// TwinCAT 3 PLC project HeatAndSteam
// ProgramVersion: 3.1.4023.0
// libraries:
//   Tc2_DataExchange, * (Beckhoff Automation GmbH)
//   Tc2_EtherCAT, * (Beckhoff Automation GmbH)
//   Tc2_MDP, * (Beckhoff Automation GmbH)
//   Tc2_ModbusSrv, * (Beckhoff Automation GmbH)
//   Tc2_Standard, * (Beckhoff Automation GmbH)
//   Tc2_SUPS, * (Beckhoff Automation GmbH)
//   Tc2_System, * (Beckhoff Automation GmbH)
//   Tc2_Utilities, * (Beckhoff Automation GmbH)
//   Tc3_DynamicMemory, * (Beckhoff Automation GmbH)
//   Tc3_EventLogger, * (Beckhoff Automation GmbH)
//   Tc3_Module, * (Beckhoff Automation GmbH)
//   Tc3_PackML_V2, * (Beckhoff Automation GmbH)
//   Tc3_PLCopen_OpcUa, * (Beckhoff Automation GmbH)
// project tree:
//   ECC/Basic/ADS Comm/ E_ADS_Comm_State.TcDUT, E_ADS_Comm_Type.TcDUT, FB_ADS_Comm.TcPOU
//   ECC/Basic/Cell/ FB_Cell_Basic.TcPOU, FB_PLC_Basic.TcPOU
//   ECC/Basic/Common Units/ E_Units.TcDUT, FB_Units.TcPOU
//   ECC/Basic/ GVL_BASIC.TcGVL
//   ECC/Basic/OPC Data/ E_StationJobData.TcDUT, F_NewDeviceDataX.TcPOU, ST_InputHeader.TcDUT, ST_OutputHeaderCellInformationX.TcDUT, ST_OutputHeaderMetaInformationX.TcDUT
//   ECC/Basic/OPC Data/Sub/ E_AlarmCategory.TcDUT, E_PML_Command.TcDUT, E_PML_Mode.TcDUT, E_PML_State.TcDUT, MaterialDataX.TcDUT, MaterialXMapping.TcDUT, ST_DataPointX.TcDUT, ST_DeviceDataX.TcDUT, ST_ErrorWarningDataX.TcDUT, ST_ManipulateMLX.TcDUT, ST_MaterialDataX.TcDUT, ST_OutputHeaderCellInformationStationInformationOperationInformationX.TcDUT, ST_OutputHeaderCellInformationStationX.TcDUT, ST_OutputHeaderTransportInformationX.TcDUT, ST_SKURestriction.TcDUT, ST_ToolDataX.TcDUT, ToolDataX.TcDUT, ToolX.TcDUT, ToolXMapping.TcDUT
//   ECC/Basic/OPC Data/Sub/Input/ ST_InputModeState.TcDUT
//   ECC/Basic/OPC Data/Sub/Output/ ST_Energy.TcDUT, ST_Exhaust.TcDUT, ST_Fluid.TcDUT, ST_JobDataOut.TcDUT, ST_OperationalDataOPxxxxx.TcDUT, ST_OutputErrorWarning.TcDUT, ST_OutputModeState.TcDUT, ST_OutputOEE.TcDUT
//   ECC/Basic/Station/ FB_Station_Basic.TcPOU
//   ECC/Basic/TrackClient/DUT/ E_CellType.TcDUT, E_MMDirection.TcTLEO, E_MMStationBuffer.TcTLEO, E_MMTrafficLightColor.TcTLEO, E_MMVehicleCommand.TcTLEO, E_MMVehicleInputType.TcTLEO, ST_MethodArgumentData.TcDUT, ST_MMBuffer.TcDUT, ST_MMLocation.TcDUT, ST_MMStation.TcDUT, ST_MMVehicleFlagData.TcDUT, ST_MMVehicleStatusData.TcDUT, ST_OPCUA_MethodData.TcDUT
//   ECC/Basic/TrackClient/Enums/ E_CarrierStatus.TcDUT, E_MMPathMotionStatus.TcTLEO, E_MMPathState.TcTLEO, E_MMServerStatus.TcTLEO, E_OPC_UA_Errors.TcDUT, E_TrackClientState.TcDUT, E_TrackState.TcDUT, E_VehicleMoveState.TcDUT
//   ECC/Basic/TrackClient/ E_CommandDataState.TcDUT, E_MappingDataState.TcDUT, E_ReworkDataState.TcDUT, FB_TrackClient_Basic.TcPOU
//   ECC/Basic/TrackClient/GVLs/ GlobalConstants.TcGVL
//   ECC/Basic/TrackClient/Method Data/Cell/ ST_GetCellIndexData.TcDUT, ST_GetCellIndexDataIn.TcDUT, ST_GetCellIndexDataOut.TcDUT
//   ECC/Basic/TrackClient/Method Data/Data/ E_MaterialType.TcDUT, E_ToolType.TcDUT, ST_AddReservationData.TcDUT, ST_AddReservationDataIn.TcDUT, ST_AddReservationDataOut.TcDUT, ST_RemoveReservationData.TcDUT, ST_RemoveReservationDataIn.TcDUT, ST_RemoveReservationDataOut.TcDUT, ST_UpdateStationBufferData.TcDUT, ST_UpdateStationBufferDataIn.TcDUT, ST_UpdateStationBufferDataOut.TcDUT, ST_UpdateVehicleDataData.TcDUT (excluded from build), ST_UpdateVehicleDataDataIn.TcDUT (excluded from build), ST_UpdateVehicleDataDataOut.TcDUT (excluded from build), ST_UpdateVehicleMappingDataData.TcDUT, ST_UpdateVehicleMappingDataDataIn.TcDUT, ST_UpdateVehicleMappingDataDataOut.TcDUT, ST_UpdateVehicleMontageData.TcDUT, ST_UpdateVehicleMontageDataIn.TcDUT, ST_UpdateVehicleMontageDataOut.TcDUT, ST_UpdateVehicleOwnerData.TcDUT, ST_UpdateVehicleOwnerDataIn.TcDUT, ST_UpdateVehicleOwnerDataOut.TcDUT, ST_UpdateVehicleReservationDataData.TcDUT, ST_UpdateVehicleReservationDataDataIn.TcDUT, ST_UpdateVehicleReservationDataDataOut.TcDUT, ST_UpdateVehicleReworkDataData.TcDUT, ST_UpdateVehicleReworkDataDataIn.TcDUT, ST_UpdateVehicleReworkDataDataOut.TcDUT
//   ECC/Basic/TrackClient/Method Data/MoveVehicle/ ST_MoveToBufferData.TcDUT, ST_MoveToBufferDataIn.TcDUT, ST_MoveToBufferDataOut.TcDUT, ST_MoveToDecisionPointData.TcDUT, ST_MoveToDecisionPointDataIn.TcDUT, ST_MoveToDecisionPointDataOut.TcDUT, ST_MoveToPositionData.TcDUT, ST_MoveToPositionDataIn.TcDUT, ST_MoveToPositionDataOut.TcDUT, ST_MoveToScannerData.TcDUT, ST_MoveToScannerDataIn.TcDUT, ST_MoveToScannerDataOut.TcDUT, ST_MoveToStationDataIn.TcDUT, ST_MoveToStationDataOut.TcDUT, ST_MoveToStationInData.TcDUT, ST_MoveToStationOutData.TcDUT, ST_MoveVehicleStatusData.TcDUT, ST_MoveVehicleStatusDataIn.TcDUT, ST_MoveVehicleStatusDataOut.TcDUT
//   ECC/Basic/TrackClient/Method Data/Path/ ST_AddPathData.TcDUT, ST_AddPathDataIn.TcDUT, ST_AddPathDataOut.TcDUT, ST_RemovePathData.TcDUT, ST_RemovePathDataIn.TcDUT, ST_RemovePathDataOut.TcDUT, ST_ResetPathData.TcDUT, ST_ResetPathDataIn.TcDUT, ST_ResetPathDataOut.TcDUT, ST_ResumePathData.TcDUT, ST_ResumePathDataIn.TcDUT, ST_ResumePathDataOut.TcDUT, ST_StartPathData.TcDUT, ST_StartPathDataIn.TcDUT, ST_StartPathDataOut.TcDUT, ST_SuspendPathData.TcDUT, ST_SuspendPathDataIn.TcDUT, ST_SuspendPathDataOut.TcDUT
//   ECC/Basic/TrackClient/Method Data/Segment/ ST_AddPathSegmentData.TcDUT, ST_AddPathSegmentDataIn.TcDUT, ST_AddPathSegmentDataOut.TcDUT, ST_GetPathSegmentVehicleCountData.TcDUT, ST_GetPathSegmentVehicleCountDataIn.TcDUT, ST_GetPathSegmentVehicleCountDataOut.TcDUT, ST_RemovePathSegmentData.TcDUT, ST_RemovePathSegmentDataIn.TcDUT, ST_RemovePathSegmentDataOut.TcDUT
//   ECC/Basic/TrackClient/Method Data/Station/ ST_AddStationData.TcDUT, ST_AddStationDataIn.TcDUT, ST_AddStationDataOut.TcDUT, ST_AddStationDoubleData.TcDUT, ST_AddStationDoubleDataIn.TcDUT, ST_AddStationDoubleDataOut.TcDUT, ST_AddStationSingleData.TcDUT, ST_AddStationSingleDataIn.TcDUT, ST_AddStationSingleDataOut.TcDUT, ST_AdjustBufferPosData.TcDUT, ST_AdjustBufferPosDataIn.TcDUT, ST_AdjustBufferPosDataOut.TcDUT, ST_EnableStationData.TcDUT, ST_EnableStationDataIn.TcDUT, ST_EnableStationDataOut.TcDUT, ST_RemoveStationData.TcDUT, ST_RemoveStationDataIn.TcDUT, ST_RemoveStationDataOut.TcDUT
//   ECC/Basic/TrackClient/Method Data/TrafficLight/ ST_AddTrafficLightData.TcDUT, ST_AddTrafficLightDataIn.TcDUT, ST_AddTrafficLightDataOut.TcDUT, ST_RemoveTrafficLightData.TcDUT, ST_RemoveTrafficLightDataIn.TcDUT, ST_RemoveTrafficLightDataOut.TcDUT, ST_SetTrafficLightColorData.TcDUT, ST_SetTrafficLightColorDataIn.TcDUT, ST_SetTrafficLightColorDataOut.TcDUT, ST_TrafficLightColorData.TcDUT, ST_TrafficLightColorDataIn.TcDUT, ST_TrafficLightColorDataOut.TcDUT
//   ECC/Basic/TrackClient/Node Data/ E_OPC_NodeType.TcDUT, ST_ReadCellData.TcDUT, ST_ReadNodeData.TcDUT, ST_ReadPathData.TcDUT, ST_ReadPathData_OLD.TcDUT, ST_ReadStationData.TcDUT, ST_ReadVehicleData.TcDUT, ST_ReadVehicleData_OLD.TcDUT, ST_StatusCell.TcDUT, ST_StatusNode.TcDUT, ST_StatusPath.TcDUT, ST_StatusStation.TcDUT, ST_StatusVehicle.TcDUT
//   ECC/Basic/TrackClient/Node Data/SUB/ ST_ReservationData.TcDUT
//   ECC/Basic/TrackClient/OPC Data/ ST_InputTransport.TcDUT, ST_OutputTransport.TcDUT
//   ECC/Basic/TrackClient/OPC Data/Sub/ ST_BufferIndexX.TcDUT, ST_CarrierX.TcDUT, ST_InputTransportAdditionalData.TcDUT, ST_InputTransportAdditionalDataMESHandShake.TcDUT, ST_InputTransportAdditionalDataSettings.TcDUT, ST_InputTransportCommand.TcDUT, ST_InputTransportConfiguration.TcDUT, ST_InputTransportMapping.TcDUT, ST_OutputTransportAdditionalData.TcDUT, ST_OutputTransportConfiguration.TcDUT, ST_OutputTransportMapping.TcDUT, ST_OutputTransportStatus.TcDUT, ST_StationBufferStatus.TcDUT, ST_StationBufferX.TcDUT, ST_StationConfigX.TcDUT, ST_StatusBuffer.TcDUT, ST_TrackLocation.TcDUT, ST_TransportMappingCarrier.TcDUT, ST_TransportMappingStationBuffer.TcDUT
//   ECC/Cell_Unit_4/ E_VehicleOnStation.TcDUT, FB_Cell_Unit_4.TcPOU, FB_OPC_Cell_Unit_4.TcPOU, ST_VehicleInHS.TcDUT
//   ECC/Cell_Unit_4/HeatAndSteamDeviceDriver/ FB_EMS_HS.TcPOU, U_EMS_HS_Read.TcDUT, U_EMS_HS_Write.TcDUT
//   ECC/Cell_Unit_4/HeatAndSteamDeviceDriver/Sub/ E_EMS_HS_Status.TcDUT, ST_EMS_HS_Alarms.TcDUT, ST_EMS_HS_Command.TcDUT, ST_EMS_HS_Read.TcDUT, ST_EMS_HS_States.TcDUT, ST_EMS_HS_Write.TcDUT
//   ECC/Cell_Unit_4/HeatAndSteam/ FB_HeatAndSteamOUT.TcPOU, F_CalcValuesHeatSteam.TcPOU, stStationVehicleCmdOut.TcDUT, E_HSStationINSeq.TcDUT, FB_HeatAndSteamIN.TcPOU
//   ECC/Cell_Unit_4/HeatAndSteam/OPC Data/Sub/AdditionalData/ ST_InputStationHSAdditionalDataOP11600.TcDUT, ST_InputStationHSAdditionalDataOP11601.TcDUT, ST_InputStationHSAdditionalDataMESHandShake.TcDUT, ST_InputStationHSAdditionalDataSettings.TcDUT, ST_OuputStationHSAdditionalDataOP11600.TcDUT, ST_OuputStationHSAdditionalDataOP11601.TcDUT, ST_InputStationHSAdditionalData.TcDUT, ST_InputStationHSAdditionalDataGeneral.TcDUT, ST_OutputStationHSAdditionalData.TcDUT, ST_OutputStationHSAdditionalDataGeneral.TcDUT
//   ECC/Cell_Unit_4/HeatAndSteam/OPC Data/Sub/Configuration/ ST_InputStationHSConfigurationOP11600.TcDUT, ST_InputStationHSUpcomingConfigurationOP11601.TcDUT, ST_InputStationHSConfigurationOP11601.TcDUT, ST_OutputStationHSCurrentConfigurationOP11601.TcDUT, ST_OutputStationHSUpcomingConfigurationOP11601.TcDUT, ST_InputStationHSConfiguration.TcDUT, ST_InputStationHSConfigurationGeneral.TcDUT, ST_InputStationHSUpcomingConfiguration.TcDUT, ST_InputStationHSUpcomingConfigurationOP11600.TcDUT, ST_OutputStationHSConfigurationOP11600.TcDUT, ST_OutputStationHSCurrentConfiguration.TcDUT, ST_OutputStationHSCurrentConfigurationGeneral.TcDUT, ST_OutputStationHSCurrentConfigurationOP11600.TcDUT, ST_OutputStationHSUpcomingConfiguration.TcDUT, ST_OutputStationHSUpcomingConfigurationOP11600.TcDUT
//   ECC/Cell_Unit_4/HeatAndSteam/OPC Data/Sub/Control/ ST_InputStationHSControlOP11601.TcDUT, ST_InputStationHSControl.TcDUT, ST_InputStationHSControlGeneral.TcDUT, ST_InputStationHSControlOP11600.TcDUT
//   ECC/Cell_Unit_4/HeatAndSteam/OPC Data/Sub/JobData/ ST_OutputStationHSJobDataOP11600.TcDUT, ST_InputStationHSJobDataOP11601.TcDUT, ST_OutputStationHSJobDataOP11601.TcDUT, ST_InputStationHSJobData.TcDUT, ST_InputStationHSJobDataOP11600.TcDUT, ST_OutputStationHSJobData.TcDUT
//   ECC/Cell_Unit_4/HeatAndSteam/OPC Data/Sub/OperationalData/ ST_OutputStationHSOperationalDataOP11601.TcDUT, ST_OutputStationHSOperationalData.TcDUT, ST_OutputStationHSOperationalDataGeneral.TcDUT, ST_OutputStationHSOperationalDataOP11600.TcDUT
//   ECC/Cell_Unit_4/OPC Data/ ST_Input.TcDUT, ST_Output.TcDUT
//   ECC/Cell_Unit_4/OPC Data/Sub/ ST_InputCell.TcDUT, ST_InputCellAdditionalData.TcDUT, ST_InputCellAdditionalDataMESHandShake.TcDUT, ST_InputCellAdditionalDataSettings.TcDUT, ST_InputCellConfiguration.TcDUT, ST_InputCellConfigurationGeneral.TcDUT, ST_InputCellControl.TcDUT, ST_InputStation.TcDUT, ST_OutputCell.TcDUT, ST_OutputCellAdditionalData.TcDUT, ST_OutputCellConfiguration.TcDUT, ST_OutputCellConfigurationGeneral.TcDUT, ST_OutputCellOperationalData.TcDUT, ST_OutputCellSustainabilityData.TcDUT, ST_OutputHeader.TcDUT, ST_OutputHeaderCellInformation.TcDUT, ST_OutputHeaderCellInformationStation.TcDUT, ST_OutputHeaderCellInformationStationInformationOperationInformation.TcDUT, ST_OutputStation.TcDUT, ST_OutputCellOperationalDataGeneral.TcDUT
//   ECC/Cell_Unit_4/HeatAndSteam/OPC Data/ ST_InputStationStationHS.TcDUT, ST_OutputStationStationHS.TcDUT
//   ECC/Cell_Unit_4/HeatAndSteam/OPC Data/Sub/Information/ ST_OutputHeaderCellInformationStationHS.TcDUT
//   ECC/Cell_Unit_4/HeatAndSteam/OPC Data/Sub/Sustainability/ ST_OutputStationHSSustainabilityData.TcDUT
//   ECC/Components/ E_ComponentErrors.TcDUT, E_Cylinder_Cmd.TcDUT, E_Cylinder_Sta.TcDUT, FB_AI.TcPOU, FB_AO.TcPOU, FB_Basic.TcPOU, FB_Blink.TcPOU, FB_Cylinder.TcPOU, FB_DI.TcPOU, FB_DO.TcPOU, FB_LIN_TRAFO.TcPOU, F_ECat_OK.TcPOU, GVL_Components.TcGVL
//   ECC/Components/TwinSAFE/ E_TwinSAFE_Group_Diag.TcDUT, E_TwinSAFE_Group_State.TcDUT, E_TwinSAFE_Logic_State.TcDUT, FB_TwinSAFE_Group.TcPOU
//   ECC/Tools/ E_Method.TcDUT, E_OPCUA_Client_Seq.TcDUT, FB_CheckHeartBeat.TcPOU, FB_GenerateHeartBeat.TcPOU, FB_GetCPULoad.TcPOU, FB_GetCPULoadPLC.TcPOU, FB_GetCPUTemp.TcPOU, FB_GetIPCSerial.TcPOU, FB_GetSafetyTemp.TcPOU, FB_GetTimePML.TcPOU, FB_OPCUA_Client_Basic.TcPOU, FB_OPCUA_Client_CallMethod.TcPOU, FB_OPCUA_Client_ReadVar.TcPOU, FB_OPCUA_GetRecipe.TcPOU, FB_OPCUA_ReadVar_BAK.TcPOU, F_Array_Sort.TcPOU, F_LogLine.TcPOU, F_StringCompNoCase.TcPOU, ST_OPC_Client_Data.TcDUT, ST_OutputArgInfoAndData_Basis.TcDUT, ST_Test.TcDUT
//   ECC/Tools/LogToFile/ FB_GetFifo.TcPOU, FB_LogToFile.TcPOU, FB_SetFifo.TcPOU, F_LogFile.TcPOU, F_PadWith.TcPOU, GVL_Log.TcGVL, ST_String_FIFO.TcDUT
//   ECC/TrackClient/Buffer Control/ FB_BufferControl.TcPOU, ST_BufferControl.TcDUT
//   ECC/TrackClient/Enums/ E_BufferState.TcDUT, E_BufferStates.TcDUT, E_PostBufferInState.TcDUT, E_DecisionPointState.TcDUT, E_ExitPointState.TcDUT, E_StationState.TcDUT, E_PostBufferOutState.TcDUT
//   ECC/TrackClient/ FB_TrackClient.TcPOU
//   ECC/TrackClient/Station Control/ E_StationBufferState.TcDUT, E_StationInOutState.TcDUT, FB_StationControl.TcPOU, ST_StationControlData.TcDUT
//   GVLs/ GVL.TcGVL
//   / PlcTask.TcTTO
//   POUs/ MAIN.TcPOU
//   ReadConfigFile/ DUT_STRUCT_VARIABLES.TcDUT, FB_ReadFile.TcPOU
// real-time tasks:
//   TASK PlcTask: cycle T#10ms, priority 20, ADS port 350
// I/O:
//   DEVICE PCI (EtherCAT) (disabled), AmsNetId 10.128.16.81.2.1
//     BusCoupler (EK1200) [EK1200-5000 EtherCAT Power supply (2A E-Bus)]
//       License (EL6070-0033) [EL6070-0033 1Ch. Licence key terminal, individual licences]
//       End (EL9011) [EL9011 End Terminal]
// variable links:
//   HeatAndSteam/HeatAndSteam Instance <-> PCI (EtherCAT)/BusCoupler (EK1200)/License (EL6070-0033)
//     PlcTask Inputs/MAIN.fbUnit4.License_AdsAdrr <-> InfoData/AdsAddr
//     PlcTask Inputs/MAIN.fbUnit4.License_State <-> InfoData/State
//     PlcTask Inputs/MAIN.fbUnit4.fbSafetyTemp.sSafetyNetID/port <-> InfoData/AdsAddr/port

CONFIGURATION HeatAndSteam
    RESOURCE PLC ON TwinCAT3
        TASK PlcTask(INTERVAL := T#10ms, PRIORITY := 20);
        PROGRAM MAIN WITH PlcTask : MAIN;
    END_RESOURCE
END_CONFIGURATION

// ---- ECC/Basic/ADS Comm/E_ADS_Comm_State.TcDUT
{attribute 'qualified_only'}
{attribute 'strict'}
TYPE E_ADS_Comm_State :
(
	Disabled := 0,
	Idle,
	Wait_Write,
	Writing,
	Write_Error,
	Wait_Read,
	Reading,
	Read_Error
);
END_TYPE

// ---- ECC/Basic/ADS Comm/E_ADS_Comm_Type.TcDUT
{attribute 'strict'}
TYPE E_ADS_Comm_Type :
(
	ADS_RD_FAST := 0,
	ADS_RD_SLOW,
	ADS_WR_FAST,
	ADS_WR_SLOW,
	ADS_RD_TRIG1,
	ADS_RD_TRIG2,
	ADS_RD_TRIG3,
	ADS_WR_TRIG1,
	ADS_WR_TRIG2,
	ADS_WR_TRIG3
);
END_TYPE

// ---- ECC/Basic/Common Units/E_Units.TcDUT
{attribute 'qualified_only'}
{attribute 'strict'}
// NOTE: Must match the array in FB_CommonUnits
TYPE E_Units :
(
	None := 0,	// 

	_m,			// Meter
	_cm,		// Centimeter
	_mm,		// Millimeter
	_um,		// Micrometer
	_nm,		// Nanometer
	
	_kg,		// Kilogram
	_g,			// Gram
	
	_RPM,		// RPM
	_mm_s,		// Millimeter pr. second
	_mm_min,	// Millimeter pr. minute
	_m_s,		// Meter pr. second
	_m_min,		// Meter pr. minute
	
	_mm_s_s,	// Millimeter pr second squared
	
	_pct,		// percent
	
	_deg,		// Degrees (angle)
	_degC,		// Degrees celcius
	_degF,		// Degrees fahrenheit
	
	_bar,		// Bar
	
	_day,		// day
	_hour,		// Hour
	_min,		// minute
	_s,			// Second
	_ms,		// Millisecond
	_us,		// Microsecond
	_ns,		// Nanosecond

	_Vac,		// Volt AC
	_Vdc,		// Volt DC
	_mV,		// Millivolt
	_a,			// Ampere
	_mA,		// Milliampere
	_uA,		// Microampere
	_KWh,		// Kilowatt hour
	_KW,		// Kilowatt
	_W,			// Watt
	_mW,		// Milliwatt
	_uW,		// Microwatt
	
	_MHz,		// Megahertz
	_kHz,		// Kilehertz
	_Hz,		// Hertz
	
	last
);
END_TYPE

// ---- ECC/Basic/OPC Data/E_StationJobData.TcDUT
{attribute 'strict'}
//
//	MAX number is 9!!
//
TYPE E_StationJobData :
(
	// Back Moulding
//	OP00100_			:= 0,

	// Brazilian Blocking
//	OP00200_			:= 0,

	// Strobeling
//	OP00300_			:= 0,

	// Manual Lasting
//	OP11400_			:= 0,

	// Automatic Lasting
//	OP11500_			:= 0,

	// Upper heat setting
//	OP11600_			:= 0,

	// Shank Placement
//	OP11700_			:= 0,

	// Ironing
//	OP11800_			:= 0,

	// Strobel Pressing
//	OP11900_			:= 0,

	// Blow Drying
//	OP12000_			:= 0,

	// Hammering
//	OP12100_			:= 0,

	// Filler Foam Placement
//	OP12200_			:= 0,

	// Manual Roughing
//	OP12300_			:= 0,

	// Robot Laser Roughing
//	OP12400_			:= 0,

	// Robot Mechanical Roughing
	OP12500_Motor 		:= 0,
	OP12500_Speed 		:= 1,
	OP12500_Pressure	:= 2,
	
	// Thread Burning
	OP12600_Heat		:= 0,
	OP12600_Air			:= 1,
	
	// Last Sorting
//	OP12700_			:= 0,

	// Last Handling
//	OP12800_			:= 0,

	// Sole Cooling
//	OP12900_			:= 0,

	// Sole Heating
//	OP13000_			:= 0,

	// Continouos Spraying
	OP13100_Color		:= 0,
	OP13100_SprayWidth	:= 1,
	OP13100_SprayPress	:= 2,
	OP13100_Tank1Press	:= 3,
	OP13100_Tank2Press	:= 4,
	
	// Burst Spraying
	OP13200_Color		:= 0,
	OP13200_SprayWidth	:= 1,
	OP13200_SprayPress	:= 2,
	OP13200_Tank1Press	:= 3,
	OP13200_Tank2Press	:= 4,
	OP13200_SprayTime	:= 5,
	OP13200_PauseTime	:= 6,

	// Sole Trimming
	OP13300_Speed		:= 0,
	OP13300_Amplitude	:= 1
	
	// Sole Buffing
//	OP13400_			:= 0,

	// Manual Delasting
//	OP13500_			:= 0,

	// Robot Delasting
//	OP13600_			:= 0,

	// Delacing
//	OP21900_			:= 0,

	// Injection
//	OP32800_			:= 0,

);
END_TYPE

// ---- ECC/Basic/OPC Data/ST_InputHeader.TcDUT
/// Standard Header for cells
TYPE ST_InputHeader :
STRUCT
	{attribute 'OPC.UA.DA.Description' := 'Header (0-100, 2 Hz)'}
	HeartBeat				: UINT;
END_STRUCT
END_TYPE

// ---- ECC/Basic/OPC Data/ST_OutputHeaderCellInformationX.TcDUT
TYPE ST_OutputHeaderCellInformationX :
STRUCT
	{attribute 'OPC.UA.DA.Description' := 'Cell name'}
	CellName				: STRING;

	{attribute 'OPC.UA.DA.Description' := 'CellID'}
	CellID					: STRING;

	{attribute 'OPC.UA.DA.Description' := 'Number of stations'}
	NumberOfStations		: UINT;

	{attribute 'OPC.UA.DA.Description' := 'Station information'}
	{attribute 'OPC.UA.DA.StructuredType' := '1'}
	TransportInformation	: ST_OutputHeaderTransportInformationX;

END_STRUCT
END_TYPE

// ---- ECC/Basic/OPC Data/ST_OutputHeaderMetaInformationX.TcDUT
TYPE ST_OutputHeaderMetaInformationX :
STRUCT
	{attribute 'OPC.UA.DA.Description' := 'Interface version'}
	InterfaceVersion		: UINT;

	{attribute 'OPC.UA.DA.Description' := 'PLC version'}
	PLCVersion				: UINT;

	{attribute 'OPC.UA.DA.Description' := 'Serial Number'}
	SerialNumber			: STRING;

	{attribute 'OPC.UA.DA.Description' := 'Cell type'}
	CellType				: STRING;

END_STRUCT
END_TYPE

// ---- ECC/Basic/OPC Data/Sub/E_AlarmCategory.TcDUT
{attribute 'qualified_only'}
TYPE E_AlarmCategory :
(
Configuration:= 1, 
Safety := 65536000,
TrackClient := 131072000,
OPCcomm := 196608000,
JobData := 262144000,
ConfigurationData := 327680000,
//GeneralSpare := 393216000,
//GeneralSpare := 458752000,
//GeneralSpare := 524288000,
//GeneralSpare := 589824000,
//GeneralSpare := 655360000,
OP11200 := 734003200,
OP11210 := 734658560,
OP11400 := 747110400,
OP11600 := 760217600,
OP11601 := 760283136,
OP11602 := 760348672,
OP11603 := 760414208,
OP11604 := 760479744,
OP11700 := 766771200,
OP12000 := 786432000,
OP12001 := 786497536,
OP12002 := 786563072,
OP12003 := 786628608,
OP12004 := 786694144,
OP12010 := 787087360,
OP12011 := 787152896,
OP12200 := 799539200,
OP12500 := 819200000,
OP12600 := 825753600,
OP12900 := 845414400,
OP12901 := 845479936,
OP12902 := 845545472,
OP12903 := 845611008,
OP12904 := 845676544,
OP12910 := 846069760,
OP12911 := 846135296,
OP12912 := 846200832,
OP12913 := 846266368,
OP12914 := 846331904,
OP13100 := 858521600,
OP13200 := 865075200,
OP13300 := 871628800,
OP13500 := 884736000,
OP13800 := 904396800,
OP16000 := 1048576000,
OP16100 := 1055129600,
OP16200 := 1061683200,
OP16300 := 1068236800,
OP16400 := 1074790400,
OP21900 := 1435238400,
OPSpare := 3276800000,
Robot := 3342336000,
LifterStation1Device := 3407872000,
LifterStation2Device := 3473408000,
LastingDevice := 3538944000
)UDINT;
END_TYPE

// ---- ECC/Basic/OPC Data/Sub/E_PML_Command.TcDUT
{attribute 'qualified_only'}
TYPE E_PML_Command :
(
	Undefined := 0,	// 0
	Reset,			// 1
	Start,			// 2
	Stop,			// 3
	Hold,			// 4
	Unhold,			// 5
	Suspend,		// 6
	Unsuspend,		// 7
	Abort,			// 8
	Clear,			// 9
	Complete		// 10
) UINT;
END_TYPE

// ---- ECC/Basic/OPC Data/Sub/E_PML_Mode.TcDUT
{attribute 'qualified_only'}
TYPE E_PML_Mode :
(
	Undefined := 0,		// Same as in E_PMLProtectedUnitMode in TC3_PackML_V2 library
	Production,			// Same as in E_PMLProtectedUnitMode in TC3_PackML_V2 library
	Maintenance,		// Same as in E_PMLProtectedUnitMode in TC3_PackML_V2 library
	Manual,				// Same as in E_PMLProtectedUnitMode in TC3_PackML_V2 library
	Calibration,		// ??
	Cleaning,			// ??
	Simulation			// Same as E_PMLProtectedUnitMode.Production, but with GVL_Components.bSIMUMode = TRUE
) UINT;
END_TYPE

// ---- ECC/Basic/OPC Data/Sub/E_PML_State.TcDUT
{attribute 'qualified_only'}
TYPE E_PML_State :
(
	Undefined := 0,	// 0
	Clearing,		// 1
	Stopped,		// 2
	Starting,		// 3
	Idle,			// 4
	Suspended,		// 5
	Execute,		// 6
	Stopping,		// 7
	Aborting,		// 8
	Aborted,		// 9
	Holding,		// 10
	Held,			// 11
	Unholding,		// 12
	Suspending,		// 13
	Unsuspending,	// 14
	Resetting,		// 15
	Completing,		// 16
	Complete		// 17
) UINT;
END_TYPE

// ---- ECC/Basic/OPC Data/Sub/Input/ST_InputModeState.TcDUT
TYPE ST_InputModeState :
STRUCT
	{attribute 'OPC.UA.DA.Description' := 'Change Request (0-255)'}
	ChangeRequest				: UINT;

	{attribute 'OPC.UA.DA.Description' := 'Requested mode (0-6)'}
	Mode						: UINT := E_PML_Mode.Production;

	{attribute 'OPC.UA.DA.Description' := 'Requested state (0-3,6,7,9'}
	State						: UINT;

END_STRUCT
END_TYPE

// ---- ECC/Basic/OPC Data/Sub/MaterialDataX.TcDUT
TYPE MaterialDataX :
STRUCT
	{attribute 'OPC.UA.DA.Description' := 'Type ID of material'}
	MaterialTypeID				: STRING(30);

	{attribute 'OPC.UA.DA.Description' := 'ID of location for material'}
	Location					: UINT;

	{attribute 'OPC.UA.DA.Description' := 'Indicator for material empty'}
	MaterialEmpty				: BOOL;

	{attribute 'OPC.UA.DA.Description' := 'Indicator for remaining material (%)'}
	MaterialRemaining			: BOOL;

END_STRUCT
END_TYPE

// ---- ECC/Basic/OPC Data/Sub/MaterialXMapping.TcDUT
TYPE MaterialXMapping :
STRUCT
	{attribute 'OPC.UA.DA.Description' := 'Type ID of material'}
	MaterialTypeID				: STRING(30);

	{attribute 'OPC.UA.DA.Description' := 'Location material is configured on'}
	Location					: UINT;

END_STRUCT
END_TYPE

// ---- ECC/Basic/OPC Data/Sub/Output/ST_Energy.TcDUT
TYPE ST_Energy :
STRUCT
END_STRUCT
END_TYPE

// ---- ECC/Basic/OPC Data/Sub/Output/ST_Exhaust.TcDUT
TYPE ST_Exhaust :
STRUCT
END_STRUCT
END_TYPE

// ---- ECC/Basic/OPC Data/Sub/Output/ST_Fluid.TcDUT
TYPE ST_Fluid :
STRUCT
END_STRUCT
END_TYPE

// ---- ECC/Basic/OPC Data/Sub/Output/ST_JobDataOut.TcDUT
TYPE ST_JobDataOut :
STRUCT
	{attribute 'OPC.UA.DA.Description' := 'Change Request (0-255)'}
	ChangeStatus				: UINT;
	
	{attribute 'OPC.UA.DA.Description' := 'Job data type'}
	JobDataType					: STRING(7);

	{attribute 'OPC.UA.DA.Description' := 'Job state (0: Undefined, 1: Idle, 2: Executing, 3: Completed'}
	JobState					: UINT;

END_STRUCT
END_TYPE

// ---- ECC/Basic/OPC Data/Sub/Output/ST_OperationalDataOPxxxxx.TcDUT
TYPE ST_OperationalDataOPxxxxx :
STRUCT
	{attribute 'OPC.UA.DA.Description' := 'Current number of tools where data is available'}
	NumberOfToolData			: UINT;

	{attribute 'OPC.UA.DA.Description' := 'Status variables for current operational data of tools'}
	{attribute 'OPC.UA.DA.StructuredType' := '1'}
	ToolData					: ARRAY [1..200] OF ToolDataX;

	{attribute 'OPC.UA.DA.Description' := 'Current number OF feeding material where data is available'}
	NumberOfMaterialData		: UINT;

	{attribute 'OPC.UA.DA.Description' := 'Status variables for current operational data of material'}
	{attribute 'OPC.UA.DA.StructuredType' := '1'}
	MaterialData				: ARRAY [1..200] OF MaterialDataX;

	{attribute 'OPC.UA.DA.Description' := 'Status variables for current operational data of devices'}
	{attribute 'OPC.UA.DA.StructuredType' := '1'}
	DeviceData					: ARRAY [1..200] OF ST_DeviceDataX;
	
END_STRUCT
END_TYPE

// ---- ECC/Basic/OPC Data/Sub/Output/ST_OutputErrorWarning.TcDUT
TYPE ST_OutputErrorWarning :
STRUCT
// Handshake part
	{attribute 'OPC.UA.DA.Description' := 'Change acknowledged (0-255)'}
	ChangeAcknowledge		: UINT;

	{attribute 'OPC.UA.DA.Description' := 'Change status (0-255)'}
	ChangeStatus			: UINT;

// Data part	
	{attribute 'OPC.UA.DA.Description' := 'Data has changed (0-65536)'}
	DataChange				: UINT;
	
	{attribute 'OPC.UA.DA.Description' := 'Current number of warnings'}
	NumberOfWarnings		: UINT;
		
	{attribute 'OPC.UA.DA.Description' := 'Current number of errors'}
	NumberOfErrors			: UINT;
	
	{attribute 'OPC.UA.DA.Description' := 'Current types of error/warnings'}
	{attribute 'OPC.UA.DA.StructuredType' := '1'}
	ErrorWarningData		: ARRAY [1..255] OF ST_ErrorWarningDataX;
	
END_STRUCT
END_TYPE

// ---- ECC/Basic/OPC Data/Sub/Output/ST_OutputModeState.TcDUT
TYPE ST_OutputModeState :
STRUCT
// Handshake part
	{attribute 'OPC.UA.DA.Description' := 'Change acknowledged (0-255)'}
	ChangeAcknowledge		: UINT;

	{attribute 'OPC.UA.DA.Description' := 'Change status (0-255)'}
	ChangeStatus			: UINT;

// Data part	
	{attribute 'OPC.UA.DA.Description' := 'Mode State data changed'}
	DataChange				: UINT;

	{attribute 'OPC.UA.DA.Description' := 'Mode State response (0-3)'}
	ModeStateResponse		: UINT;		// 0: Undefined, 1: Could not handle, 2: Request declined, 3: OK

	{attribute 'OPC.UA.DA.Description' := 'Current mode (0-6)'}
	CurrentMode				: UINT;

	{attribute 'OPC.UA.DA.Description' := 'Requested mode (0-6)'}
	RequestedMode			: UINT;

	{attribute 'OPC.UA.DA.Description' := 'Current state (0-17)'}
	CurrentState			: UINT;

	{attribute 'OPC.UA.DA.Description' := 'Requested state (0-17)'}
	RequestedState			: UINT;

END_STRUCT
END_TYPE

// ---- ECC/Basic/OPC Data/Sub/Output/ST_OutputOEE.TcDUT
TYPE ST_OutputOEE :
STRUCT
// Handshake part
	{attribute 'OPC.UA.DA.Description' := 'Change acknowledged (0-255)'}
	ChangeAcknowledge	: UINT;

	{attribute 'OPC.UA.DA.Description' := 'Change status (0-255)'}
	ChangeStatus		: UINT;

// Data part	
	{attribute 'OPC.UA.DA.Description' := 'Data has changed (0-65536)'}
	DataChange			: UINT;
	
	{attribute 'OPC.UA.DA.Description' := 'Date and time'}
	DateTime	 		: DT;
	
	{attribute 'OPC.UA.DA.Description' := ''}
	EventID		 		: UDINT;
	
	{attribute 'OPC.UA.DA.Description' := 'Counter for all processed products'}
	ProcessedProduct	: UDINT;

	{attribute 'OPC.UA.DA.Description' := 'Counter for all processed good products'}
	GoodProduct			: UDINT;

	{attribute 'OPC.UA.DA.Description' := 'Counter for all processed rejected products'}
	RejectedProduct		: UDINT;

END_STRUCT
END_TYPE

// ---- ECC/Basic/OPC Data/Sub/ST_DataPointX.TcDUT
TYPE ST_DataPointX :
STRUCT
	X					: REAL;	// Point on shoe. X value.
	Y					: REAL;	// Point on shoe. Y value.
	Z					: REAL;	// Point on shoe. Z value.
	Q1					: REAL;	// Point on shoe. Quaternion scalar part
	Q2					: REAL;	// Point on shoe. Quaternion x vector part
	Q3					: REAL;	// Point on shoe. Quaternion y vector part
	Q4					: REAL;	// Point on shoe. Quaternion z vector part
	Speed				: REAL;	// Speed setting.
	Acceleration		: REAL;	// Acceleration setting
	Zone				: REAL;	// Zone setting
//	ExternalTCP			: UINT;	// ID of external TCP. This can be referencepoints for tools or otherpoints of interests.
	ExternalTCPOffsetX	: REAL;	// External TCP offset. X value.
	ExternalTCPOffsetY	: REAL;	// External TCP offset. Y value.
	ExternalTCPOffsetZ	: REAL;	// External TCP offset. Z value.
	ExternalTCPOffsetQ1	: REAL;	// External TCP offset. Quaternion scalar part
	ExternalTCPOffsetQ2	: REAL;	// External TCP offset. Quaternion x vector part
	ExternalTCPOffsetQ3	: REAL;	// External TCP offset. Quaternion y vector part
	ExternalTCPOffsetQ4	: REAL;	// External TCP offset. Quaternion z vector part
	Validate			: BOOL;	// Indicator that a validation from the bridge is required before moving to a point. Robot will move to a safepos untill validation is recieved from the bridge
	arDeviceParameters	: ARRAY [0..9] OF REAL;	// See "E_StationJobData" for array specification

END_STRUCT
END_TYPE

// ---- ECC/Basic/OPC Data/Sub/ST_DeviceDataX.TcDUT
TYPE ST_DeviceDataX :
STRUCT
	{attribute 'OPC.UA.DA.Description' := 'The ID of the specific device'}
	DeviceID			: STRING(30);

	{attribute 'OPC.UA.DA.Description' := 'The descriptive name of the device'}
	DeviceName			: STRING(30);

	{attribute 'OPC.UA.DA.Description' := 'The ID of the operational data'}
	DataID				: UDINT;

	{attribute 'OPC.UA.DA.Description' := 'The descriptive name of the operational data'}
	DataName			: STRING(30);

	{attribute 'OPC.UA.DA.Description' := 'The value of the operational data'}
	Value				: REAL;

	{attribute 'OPC.UA.DA.Description' := 'The ID code for the measuring unit'}
	UnitID				: STRING(30);

	{attribute 'OPC.UA.DA.Description' := 'The symbolic description of the measuring unit'}
	Unit				: STRING(30);

END_STRUCT
END_TYPE

// ---- ECC/Basic/OPC Data/Sub/ST_ErrorWarningDataX.TcDUT
TYPE ST_ErrorWarningDataX :
STRUCT
	{attribute 'OPC.UA.DA.Description' := 'Error/Warning type. 0: Undefined, 1: Warning, 2: Error'}
	ErrorWarningType	: UINT;
	
	{attribute 'OPC.UA.DA.Description' := 'Cell ID or Station ID'}
	LocationID			: STRING(30);
	
	{attribute 'OPC.UA.DA.Description' := 'Trigger data and time'}
	DateTime			: STRING;	

	{attribute 'OPC.UA.DA.Description' := 'ID of the error/warning'}
	ErrorWarningID		: UDINT;	

	{attribute 'OPC.UA.DA.Description' := 'ID of the specific device/tool (optional)'}
	DeviceID			: STRING(30);	

	{attribute 'OPC.UA.DA.Description' := 'Severity of the event. 0: Undefined, 1: Low, 2: High'}
	Severity			: UINT;	

	{attribute 'OPC.UA.DA.Description' := 'ID from the native device'}
	NativeID			: UDINT;	

	{attribute 'OPC.UA.DA.Description' := 'Message from the native device'}
	NativeMessage		: STRING(80);	

END_STRUCT
END_TYPE

// ---- ECC/Basic/OPC Data/Sub/ST_ManipulateMLX.TcDUT
TYPE ST_ManipulateMLX :
STRUCT
	iNumberOfDataPoint		: USINT;			// Indicator for how many OF the data points that are filled out.
	ScaleOriginX 			: REAL;				// Origin of scale point. X value.
	ScaleOriginY			: REAL;				// Origin of scale point. Y value.
	ScaleOriginZ			: REAL;				// Origin of scale point. Z value.
	ScaleOriginQ1			: REAL;				// Origin of scale point. Quaternion scalar part
	ScaleOriginQ2			: REAL;				// Origin of scale point. Quaternion x vector part
	ScaleOriginQ3			: REAL;				// Origin of scale point. Quaternion y vector part
	ScaleOriginQ4			: REAL;				// Origin of scale point. Quaternion z vector part
	ScaleFactorX			: REAL;				// Scale factor in x direction.
	ScaleFactorYZ			: REAL;				// Scale factor in y and z direction.
	CalibrationOffsetX		: REAL;				// Offset from calibration of machine last. X value.
	CalibrationOffsetY		: REAL;				// Offset from calibration of machine last. Y value.
	CalibrationOffsetZ		: REAL;				// Offset from calibration of machine last. Z value.
	CalibrationOffsetQ1		: REAL;				// Offset from calibration of machine last. Quaternion scalar part
	CalibrationOffsetQ2		: REAL;				// Offset from calibration of machine last. Quaternion x vector part
	CalibrationOffsetQ3		: REAL;				// Offset from calibration of shoe last. Quaternion y vector part
	CalibrationOffsetQ4		: REAL;				// Offset FROM calibration OF shoe last. Quaternion z vector part	
	aDataPoints				: ARRAY [0..199] OF ST_DataPointX;// Parameters for first point on shoe/machine last.
END_STRUCT
END_TYPE

// ---- ECC/Basic/OPC Data/Sub/ST_MaterialDataX.TcDUT
TYPE ST_MaterialDataX :
STRUCT
	{attribute 'OPC.UA.DA.Description' := 'Job data type'}

END_STRUCT
END_TYPE

// ---- ECC/Basic/OPC Data/Sub/ST_OutputHeaderCellInformationStationInformationOperationInformationX.TcDUT
TYPE ST_OutputHeaderCellInformationStationInformationOperationInformationX :
STRUCT
	{attribute 'OPC.UA.DA.Description' := 'Operation name'}
	OperationName			: STRING;

	{attribute 'OPC.UA.DA.Description' := 'Operation ID'}
	OperationID				: STRING;

END_STRUCT
END_TYPE

// ---- ECC/Basic/OPC Data/Sub/ST_OutputHeaderCellInformationStationX.TcDUT
TYPE ST_OutputHeaderCellInformationStationX :
STRUCT
	{attribute 'OPC.UA.DA.Description' := 'Station name'}
	StationName				: STRING;

	{attribute 'OPC.UA.DA.Description' := 'Station ID'}
	StationID				: STRING;
	
	{attribute 'OPC.UA.DA.Description' := 'PLC version'}
	NumberOfOperations		: UINT;
	
	{attribute 'OPC.UA.DA.Description' := 'Rework possible on this station'}
	Rework					: BOOL;

END_STRUCT
END_TYPE

// ---- ECC/Basic/OPC Data/Sub/ST_OutputHeaderTransportInformationX.TcDUT
TYPE ST_OutputHeaderTransportInformationX :
STRUCT
	{attribute 'OPC.UA.DA.Description' := 'Transport name'}
	TransportName			: STRING;

	{attribute 'OPC.UA.DA.Description' := 'Transport type'}
	TransportType			: STRING;
	
END_STRUCT
END_TYPE

// ---- ECC/Basic/OPC Data/Sub/ST_SKURestriction.TcDUT
TYPE ST_SKURestriction :
STRUCT
	{attribute 'OPC.UA.DA.Description' := 'TRUE of restrictions are active'}
	Restricted				: BOOL;

	{attribute 'OPC.UA.DA.Description' := 'Number of defined SKU restrictions (0-200)'}
	NumberOfRestrictions	: UINT;
	
	{attribute 'OPC.UA.DA.Description' := 'ID of SKUs that the operation is restricted to handle'}
	SKUID					: ARRAY [1..200] OF STRING(30);
	
END_STRUCT
END_TYPE

// ---- ECC/Basic/OPC Data/Sub/ST_ToolDataX.TcDUT
TYPE ST_ToolDataX :
STRUCT
	{attribute 'OPC.UA.DA.Description' := 'Job data type'}

END_STRUCT
END_TYPE

// ---- ECC/Basic/OPC Data/Sub/ToolDataX.TcDUT
TYPE ToolDataX :
STRUCT
	{attribute 'OPC.UA.DA.Description' := 'Unique ID of Tool'}
	TooID					: UINT;

	{attribute 'OPC.UA.DA.Description' := 'ID of the location of Tool'}
	Location				: UINT;

	{attribute 'OPC.UA.DA.Description' := 'Usage cycles since tool configuration'}
	CurrentCycles			: UDINT;

	{attribute 'OPC.UA.DA.Description' := 'Max allowed cycles for tool'}
	MaxCycles				: UDINT;

END_STRUCT
END_TYPE

// ---- ECC/Basic/OPC Data/Sub/ToolX.TcDUT
TYPE ToolX :
STRUCT
	{attribute 'OPC.UA.DA.Description' := 'Unique ID of tool'}
	ToolID					: STRING(30);
	
	{attribute 'OPC.UA.DA.Description' := 'ID for type of tool'}
	ToolTypeID				: STRING(30);

END_STRUCT
END_TYPE

// ---- ECC/Basic/OPC Data/Sub/ToolXMapping.TcDUT
TYPE ToolXMapping :
STRUCT
	{attribute 'OPC.UA.DA.Description' := 'Unique ID of tool'}
	ToolID						: STRING(30);

	{attribute 'OPC.UA.DA.Description' := 'ID for the location tool is configured on'}
	Location					: UINT;

	{attribute 'OPC.UA.DA.Description' := 'Max allowed tool cycles'}
	MaxCycles					: UINT;

END_STRUCT
END_TYPE

// ---- ECC/Basic/TrackClient/DUT/E_CellType.TcDUT
{attribute 'qualified_only'}
{attribute 'strict'}
TYPE E_CellType :
(
	Type_Outline := 0,		// Cell has own track with inlet and outlet tracks
	Type_Inline := 1,		// Cell/station is placed on the main track
	Type_InOut := 2			// Cell has only one track for handling both inlet and outlet (no queue functionality)
	
	
);
END_TYPE

// ---- ECC/Basic/TrackClient/DUT/E_MMDirection.TcTLEO
{attribute 'qualified_only'}
TYPE E_MMDirection :
(
	eMMDirection_BiDirectional	:= 0,																				(**)
	eMMDirection_Forward		:= 1,																				(**)
	eMMDirection_Backward		:= 2																				(**)
) BYTE;
END_TYPE

// ---- ECC/Basic/TrackClient/DUT/E_MMStationBuffer.TcTLEO
{attribute 'qualified_only'}
{attribute 'strict'}
TYPE E_MMStationBuffer :
(
	eMMStationBuffer_PreProcess		:= 0,
	eMMStationBuffer_PostProcess	:= 1
);
END_TYPE

// ---- ECC/Basic/TrackClient/DUT/E_MMTrafficLightColor.TcTLEO
{attribute 'qualified_only'}
TYPE E_MMTrafficLightColor :
(
	eMMTrafficLightColor_NA		:= -1,
	eMMTrafficLightColor_Green	:= 0,
	eMMTrafficLightColor_Red	:= 1
);
END_TYPE
//  eMMTrafficLightColor_NA = '-1'

// ---- ECC/Basic/TrackClient/DUT/E_MMVehicleCommand.TcTLEO
{attribute 'qualified_only'}
TYPE E_MMVehicleCommand :
(
	eMMVehicleCommand_NoCommandInProgress 	:= 0,																	(**)
	eMMVehicleCommand_MoveVehicleToStation	:= 176,																	(**)
	eMMVehicleCommand_MoveVehicleToPosition	:= 177																	(**)
) BYTE;
END_TYPE

// ---- ECC/Basic/TrackClient/DUT/E_MMVehicleInputType.TcTLEO
{attribute 'qualified_only'}
{attribute 'strict'}
TYPE E_MMVehicleInputType :
(
	eMMVehicleInputType_VehicleID			:= 0,	// MagneMotion ID
	eMMVehicleInputType_CarrierID			:= 1,	// RFID scanned ID from Carrier
	eMMVehicleInputType_LastID 				:= 2,	// RFID scanned Id from Last
	eMMVehicleInputType_ArticleID 			:= 3,
	eMMVehicleInputType_LastTypeID			:= 4,
	eMMVehicleInputType_StationID			:= 5,
	eMMVehicleInputType_CellID				:= 6,
	eMMVehicleInputType_EmptyVehicles		:= 7,
	eMMVehicleInputType_ReleasedVehicles	:= 8,
	eMMVehicleInputType_AllVehicles			:= 9
);
END_TYPE

// ---- ECC/Basic/TrackClient/DUT/ST_MethodArgumentData.TcDUT
TYPE ST_MethodArgumentData :
STRUCT
	eDataType		: E_UADataType;
	pData			: PVOID;
	nDataSize		: UINT;
	
END_STRUCT
END_TYPE

// ---- ECC/Basic/TrackClient/DUT/ST_MMBuffer.TcDUT
{attribute 'OPC.UA.DA.StructuredType':='1'}
TYPE ST_MMBuffer :
STRUCT
	bPresent					: BOOL	:= FALSE;																	(* Flag for indicating if the buffer position is present/used*)
	stLocation					: ST_MMLocation;																	(* Location of the buffer on the track. *)
	nTicket						: UINT;
	nTicketSize					: UINT;
	nReservedVehicleID			: UINT;
	nCurrentVehicleID			: UINT;
	CurrentPriority				: UINT;
//	sReservedCarrierID			: STRING(30);
//	sCurrentCarrierID			: STRING(30);
END_STRUCT
END_TYPE

// ---- ECC/Basic/TrackClient/DUT/ST_MMLocation.TcDUT
{attribute 'OPC.UA.DA.StructuredType':='1'}
TYPE ST_MMLocation :
STRUCT
	nPathID						: UINT	:= 0;		(* The path the position is related to. *)
	fPosition					: REAL	:= 0;		(* [M] The position on the path. *)
END_STRUCT
END_TYPE

// ---- ECC/Basic/TrackClient/DUT/ST_MMStation.TcDUT
{attribute 'OPC.UA.DA.StructuredType':='1'}
TYPE ST_MMStation :
STRUCT
	sCellID						: STRING := '';												(* The cell that the station belongs to. *)
	sStationID					: STRING(30) := '';											(* The identifier for the station. *)
	bPresent					: BOOL := FALSE;											(* Flag for indicating if the station is present. *)
	stStationData1				: ST_MMBuffer;												(* The location of the station. *)
	stStationData2				: ST_MMBuffer;												(* The location of the station. *)
	stDecisionLocation			: ST_MMLocation;											(* The location of the decision point of the station. *)
	astPreBuffer				: ARRAY[1..MM_MAX_BUFFER_INDEX] OF ST_MMBuffer;				(* The stations prebuffer. *)
	astPostBuffer				: ARRAY[1..MM_MAX_BUFFER_INDEX] OF ST_MMBuffer;				(* The stations postbuffer. *)
END_STRUCT
END_TYPE

// ---- ECC/Basic/TrackClient/DUT/ST_MMVehicleFlagData.TcDUT
TYPE ST_MMVehicleFlagData :
STRUCT
	bVehicleSignal				: BOOL;
	bObstructedStatus			: BOOL;
	bHinderedStatus				: BOOL;
	nPIDLoopSetIndex			: USINT;
	bSuspectStatus				: BOOL;
END_STRUCT
END_TYPE

// ---- ECC/Basic/TrackClient/DUT/ST_MMVehicleStatusData.TcDUT
TYPE ST_MMVehicleStatusData :
STRUCT
	nVehicleID					: UINT;
	bVehiclePresent				: BOOL;
	nPathID						: UINT;
	nDestinationPathID			: UINT;
	fVehiclePosition			: REAL;
	fVelocity					: REAL;
	eVehicleCommandType			: E_MMVehicleCommand;
	stVehicleFlags				: ST_MMVehicleFlagData;
	fVehicleCommandedPosition	: REAL;
	nVehicleCommandedStation	: USINT;
END_STRUCT
END_TYPE

// ---- ECC/Basic/TrackClient/DUT/ST_OPCUA_MethodData.TcDUT
// Data needed for OPC UA method calling
TYPE ST_OPCUA_MethodData :
STRUCT
	bActivate						: BOOL;		// TRUE to use this method call

	// Method information:
	sRemoteObjectName				: STRING;	// Remote object. e.g. 'MAIN.fbMMServer'
	sRemoteMethodName				: STRING;	// Remote method. e.g. 'M_AddPath'

	// Input data:
	NoOfInputArgs					: BYTE;		// Number of input arguments for the remote method
	
	
	// Output data:
	NoOfOutputArgs					: BYTE;		// Number of output arguments for the remote method
	
	
END_STRUCT
END_TYPE

// ---- ECC/Basic/TrackClient/Enums/E_CarrierStatus.TcDUT
{attribute 'qualified_only'}
{attribute 'strict'}
TYPE E_CarrierStatus :
(
	Undefined := 0,			// Recently discovered, not scanned or assigned to anything
	Initiating,				// On the way to scanning
	NotBusy,				// Not assigned to a job
	Busy,					// Assigned to a job
	MontageReserved			// Reserved for a tool, but tool is removed temporarily (must be free to mount same tool again)

);
END_TYPE

// ---- ECC/Basic/TrackClient/Enums/E_MMPathMotionStatus.TcTLEO
{attribute 'qualified_only'}
TYPE E_MMPathMotionStatus :
(
	eMMPathMotionStatus_Enabled				:= 0,																	(**)
	eMMPathMotionStatus_SuspendedByCommand	:= 1,																	(**)
	eMMPathMotionStatus_EStopActive			:= 2,																	(**)
	eMMPathMotionStatus_InterlockActive		:= 3																	(**)
) BYTE;
END_TYPE

// ---- ECC/Basic/TrackClient/Enums/E_MMPathState.TcTLEO
{attribute 'qualified_only'}
TYPE E_MMPathState :
(
	eMMPathState_Initialization 		:= 0,																		(**)
	eMMPathState_Startup				:= 1,																		(**)
	eMMPathState_Operational			:= 2,																		(**)
	eMMPathState_ResetInProgress		:= 3,																		(**)
	eMMPathState_ProgrammingInProgress	:= 4																		(**)
) BYTE;
END_TYPE

// ---- ECC/Basic/TrackClient/Enums/E_MMServerStatus.TcTLEO
{attribute 'qualified_only'}
{attribute 'strict'}
TYPE E_MMServerStatus :
(
	eMMServerStatus_Default										:= 0,
	eMMServerStatus_Success										:= 1,
	eMMServerStatus_Rejected_UserInputError						:= 2,
	eMMServerStatus_Rejected_NotAllowed							:= 3,
	eMMServerStatus_Rejected_ConfigurationAlreadyDefined		:= 20,
	eMMServerStatus_Rejected_NotDefinedInConfiguration			:= 21,
	eMMServerStatus_Rejected_VehicleRelatedInfoNotFound			:= 40,
	eMMServerStatus_Failed_UnableToRemoveFromConfiguration		:= 100,
	eMMServerStatus_Failed_CouldNotHandleMoveVehicleRequest		:= 120
);
END_TYPE

// ---- ECC/Basic/TrackClient/Enums/E_OPC_UA_Errors.TcDUT
{attribute 'qualified_only'}
TYPE E_OPC_UA_Errors :
(
	NO_ERROR						:= 16#00000000, // No error
	DEVICE_INVALIDSIZE				:= 16#00000705, // Parameter size not correct
	DEVICE_INVALIDDATA				:= 16#00000706, // Invalid parameter values
	DEVICE_NOMEMORY					:= 16#0000070A, // Not enough memory

	UAC_E_FAIL						:= 16#E4DD0001, // UA service call failed
	UAC_E_CONNECTED					:= 16#E4DD0100, // Server already connected
	UAC_E_CONNECT					:= 16#E4DD0101, // General error when establishing a connection
	UAC_E_UASECURITY				:= 16#E4DD0102, // UA security could not be set up
	UAC_E_ITEMEXISTS				:= 16#E4DD0103, // Element ID already exists
	UAC_E_ITEMNOTFOUND				:= 16#E4DD0104, // Element does not exist
	UAC_E_ITEMTYPE					:= 16#E4DD0105, // Invalid or unsupported item type
	UAC_E_CONVERSION				:= 16#E4DD0106, // Variable types cannot be converted
	UAC_E_SUSPENDED					:= 16#E4DD0107, // Device hangs. Please try again later...
	UAC_E_TYPE_NOT_SUPPORTED		:= 16#E4DD0108, // Conversion variable type is not supported.
	UAC_E_NSNAME_NOTFOUND			:= 16#E4DD0109, // No namespace with the specified name found.
	UAC_E_CONNECT_NOTFOUND			:= 16#E4DD0110, // Connection failed: Target host could not be found.
	UAC_E_TIMEOUT					:= 16#E4DD0111, // Timeout: i.e. target host does not respond
	UAC_E_INVALIDHDL				:= 16#E4DD0112, // Session handle invalid
	UAC_E_INVALIDNODEID				:= 16#E4DD0113, // UA node ID unknown
	UAC_E_INVAL_IDENTIFIER_TYPE		:= 16#E4DD0114, // Identifier type of UaNodeId invalid
	UAC_E_IDENTIFIER_NOTSUPP		:= 16#E4DD0115, // Identifier type UaNodeId is not supported
	UAC_E_INVAL_NODE_HDL			:= 16#E4DD0116, // Invalid node handle
	UAC_E_UAREADFAILED				:= 16#E4DD0117, // UA read failed for unknown reasons
	UAC_E_UAWRITEFAILED				:= 16#E4DD0118, // UA write failed for unknown reasons
	UAC_E_INVAL_NODEMETHOD_HDL		:= 16#E4DD0119, // Invalid method handle
	UAC_E_CALL_FAILED				:= 16#E4DD011A, // Call failed, cause unknown
	UAC_E_CALLDECODE_FAILED			:= 16#E4DD011B, // Successful call, decoding return value failed
	UAC_E_NOTMAPPEDTYPE				:= 16#E4DD011C, // Unassigned data type in return value
	UAC_E_CALL_FAILED_BADINTERNAL	:= 16#E4DD011D, // Call failed with UA_BadInternal
	UAC_E_METHODIDINVALID			:= 16#E4DD011E, // Unknown MethodID (returned on call, even if provided by GetMethodHdl)
	UAC_E_TOOMUCHDIM				:= 16#E4DD011F, // Method call has returned parameters with more than 3 dimensions; not supported.
	UAC_E_CALL_FAILED_INVALIDARG	:= 16#E4DD0120, // Call failed with OpcUa_BadInvalidArgument
	UAC_E_CALL_FAILED_TYPEMISMATCH	:= 16#E4DD0121, // Call failed with UAC_E_CALL_FAILED_TYPEMISMATCH
	UAC_E_CALL_FAILED_OUTOFRANGE	:= 16#E4DD0122, // Call failed with UAC_E_CALL_FAILED_OUTOFRANGE
	UAC_E_CALL_FAILED_BADSTRUCTURE	:= 16#E4DD0123, // Call failed with OpcUa_BadStructureMissing
	UAC_E_CALL_TYPEMISMATCH_OUTPARAM:= 16#E4DD0124, // Call successful, but type of output information provided does not match
	UAC_E_NONVALIDTYPEINFO			:= 16#E4DD0125, // Node has insufficient type information
	UAC_E_INVALIDATTRIBID			:= 16#E4DD0126, // Access to invalid node attribute
	UAC_E_NOTSUPPORTED				:= 16#E4DD0128, // The command is not supported by the connected UaServer, e.g. when calling UA_HistoryUpdate.
	UAC_E_INVALID_ARRAY_LENGTH		:= 16#E4DE0100, // An invalid array length not matching DataValueCount was assigned to UA_HistoryUpdate.
	UAC_E_INVALID_DATASIZE			:= 16#E4DE0101, // A data value with an invalid data type size was assigned to UA_HistoryUpdate. All assigned DataValues must be of the same data type.
	UAC_E_SUBERROR					:= 16#E4DE0102 // A lower-level error was output for at least one of the transferred data values. See ValueErrorIDs at UA_HistoryUpdate.
		
) UDINT;
END_TYPE

// ---- ECC/Basic/TrackClient/Enums/E_TrackClientState.TcDUT
{attribute 'qualified_only'}
{attribute 'strict'}
TYPE E_TrackClientState :
(
	Disconnected := 0,
	(* Connect *)
	Connecting,
	GetNamespaceIndex,
	Connected,
	(* Execute function *)
	GetHandle,
	Execute,
	ReleaseHandle,
	(* Disconnect *)	
	Disconnecting,
	Error
);
END_TYPE

// ---- ECC/Basic/TrackClient/Enums/E_TrackState.TcDUT
{attribute 'qualified_only'}
{attribute 'strict'}
TYPE E_TrackState :
(
	Undefined := 0,
	CheckInitDone,
//	InitDecisionPoint,
	WaitAllowInit,
	InitStations,
	SetPreBufferAdjust,
	SetPostBufferAdjust,
	InitPaths,
//	InitPathsStations,
//	InitPathsDecisionPoint,
//	InitPathsTrafficLight,
	InitGetCellIndex,
	Idle,
	Resetting,
	ResetWait,
	ResetCheck,
	Starting,
	StartCheck,
	InitTrafficLight,
	InitTrafficLight2,
	InitPathSegment,
	InitPathSegment2,
	InitVehicles,
	Started,
	Suspend,
	Suspending,
	Suspended,
	Resume,
	Resuming,
	Error
);
END_TYPE

// ---- ECC/Basic/TrackClient/Enums/E_VehicleMoveState.TcDUT
{attribute 'qualified_only'}
{attribute 'strict'}
TYPE E_VehicleMoveState :
(
	Unknown := 0,
	Idle,
	Pending,
	Accepted,
	Moving,
	Complete,
	ErrorLocation
	
);
END_TYPE

// ---- ECC/Basic/TrackClient/E_CommandDataState.TcDUT
{attribute 'qualified_only'}
{attribute 'strict'}
TYPE E_CommandDataState :
(
	Undefined := 0,
	CheckRequest,
	AddReservation,
	UpdateJobData,
	Done,
	Error
);
END_TYPE

// ---- ECC/Basic/TrackClient/E_MappingDataState.TcDUT
{attribute 'qualified_only'}
{attribute 'strict'}
TYPE E_MappingDataState :
(
	Undefined := 0,
	CheckRequest,
	UpdateMappingData,
	UpdateReworkData,
	Done,
	Error
);
END_TYPE

// ---- ECC/Basic/TrackClient/E_ReworkDataState.TcDUT
{attribute 'qualified_only'}
{attribute 'strict'}
TYPE E_ReworkDataState :
(
	Undefined := 0,
	CheckRequest,
	UpdateReworkData,
	Done,
	Error
);
END_TYPE

// ---- ECC/Basic/TrackClient/Method Data/Cell/ST_GetCellIndexData.TcDUT
TYPE ST_GetCellIndexData :
STRUCT
	sObjectID					: STRING := 'MAIN.fbMMServer';
	sMethodID					: STRING := 'MAIN.fbMMServer#M_GetCellIndex';
	iStatus						: INT;
	iNoOfInputArgs				: BYTE := 1;
	iNoOfOutputArgs				: BYTE := 3;
	stInput						: ST_GetCellIndexDataIn;
	stOutput					: ST_GetCellIndexDataOut;	
END_STRUCT
END_TYPE

// ---- ECC/Basic/TrackClient/Method Data/Cell/ST_GetCellIndexDataIn.TcDUT
{attribute 'pack_mode' := '1'}
TYPE ST_GetCellIndexDataIn :
STRUCT
	sCellID						: STRING(30);
END_STRUCT
END_TYPE

// ---- ECC/Basic/TrackClient/Method Data/Cell/ST_GetCellIndexDataOut.TcDUT
{attribute 'pack_mode' := '1'}
TYPE ST_GetCellIndexDataOut :
STRUCT
	// Fixed data for all methods
	nNumberOfOutputArguments	: UDINT;								// determined amount of output parameters
	nReserved					: ARRAY[1..4] OF BYTE;					// Reserved padding
	
	// Method specific data
	stOutputArgInfo				: ARRAY[1..3] OF ST_UAMethodArgInfo; 	//
	nCellIndex					: UINT; 								// Cell index for status structures on Track Server
	eStatus						: E_MMServerStatus;						// Status from remote method (succes/fail)
	sMessage					: STRING;								// Debugging message

END_STRUCT
END_TYPE

// ---- ECC/Basic/TrackClient/Method Data/Data/E_MaterialType.TcDUT
{attribute 'qualified_only'}
{attribute 'strict'}
TYPE E_MaterialType :
(
	Undefined := 0,
	None,
	Upper
);
END_TYPE

// ---- ECC/Basic/TrackClient/Method Data/Data/E_ToolType.TcDUT
{attribute 'qualified_only'}
{attribute 'strict'}
TYPE E_ToolType :
(
	Undefined := 0,
	None,
	Last,
	Tray
);
END_TYPE

// ---- ECC/Basic/TrackClient/Method Data/Data/ST_AddReservationData.TcDUT
TYPE ST_AddReservationData :
STRUCT
	sObjectID					: STRING := 'MAIN.fbMMServer';
	sMethodID					: STRING := 'MAIN.fbMMServer#M_AddReservationList';
	iStatus						: INT;
	iNoOfInputArgs				: BYTE := 5;
	iNoOfOutputArgs				: BYTE := 2;
	stInput						: ST_AddReservationDataIn;
	stOutput					: ST_AddReservationDataOut;	
END_STRUCT
END_TYPE

// ---- ECC/Basic/TrackClient/Method Data/Data/ST_AddReservationDataIn.TcDUT
{attribute 'pack_mode' := '1'}
TYPE ST_AddReservationDataIn :
STRUCT
	sStationID					: STRING(30);								(* The ID of the station that will be moved to. *)
	sCarrierID					: STRING(30);								(* Carrier ID of vehicle at buffer position *)
	nTicket						: UINT;										(* Ticket number *)
	nTicketSize					: UINT;										(* Ticket size (number of vehicles with same ticket) *)
	nPriority					: UINT;										(* Ticket priority *)
END_STRUCT
END_TYPE

// ---- ECC/Basic/TrackClient/Method Data/Data/ST_AddReservationDataOut.TcDUT
{attribute 'pack_mode' := '1'}
TYPE ST_AddReservationDataOut :
STRUCT
	// Fixed data for all methods
	nNumberOfOutputArguments	: UDINT;								// determined amount of output parameters
	nReserved					: ARRAY[1..4] OF BYTE;					// Reserved padding
	
	// Method specific data
	stOutputArgInfo				: ARRAY[1..2] OF ST_UAMethodArgInfo; 	// 
	eStatus						: E_MMServerStatus;						// Status from remote method (succes/fail)
	sMessage					: STRING;								// Debugging message

END_STRUCT
END_TYPE

// ---- ECC/Basic/TrackClient/Method Data/Data/ST_RemoveReservationData.TcDUT
TYPE ST_RemoveReservationData :
STRUCT
	sObjectID					: STRING := 'MAIN.fbMMServer';
	sMethodID					: STRING := 'MAIN.fbMMServer#M_RemoveReservationList';
	iStatus						: INT;
	iNoOfInputArgs				: BYTE := 2;
	iNoOfOutputArgs				: BYTE := 2;
	stInput						: ST_RemoveReservationDataIn;
	stOutput					: ST_RemoveReservationDataOut;	
END_STRUCT
END_TYPE

// ---- ECC/Basic/TrackClient/Method Data/Data/ST_RemoveReservationDataIn.TcDUT
{attribute 'pack_mode' := '1'}
TYPE ST_RemoveReservationDataIn :
STRUCT
	sStationID					: STRING(30);								(* The ID of the station that will be moved to. *)
	nTicket						: UINT;										(* Ticket number *)
END_STRUCT
END_TYPE

// ---- ECC/Basic/TrackClient/Method Data/Data/ST_RemoveReservationDataOut.TcDUT
{attribute 'pack_mode' := '1'}
TYPE ST_RemoveReservationDataOut :
STRUCT
	// Fixed data for all methods
	nNumberOfOutputArguments	: UDINT;								// determined amount of output parameters
	nReserved					: ARRAY[1..4] OF BYTE;					// Reserved padding
	
	// Method specific data
	stOutputArgInfo				: ARRAY[1..2] OF ST_UAMethodArgInfo; 	// 
	eStatus						: E_MMServerStatus;						// Status from remote method (succes/fail)
	sMessage					: STRING;								// Debugging message

END_STRUCT
END_TYPE

// ---- ECC/Basic/TrackClient/Method Data/Data/ST_UpdateStationBufferData.TcDUT
TYPE ST_UpdateStationBufferData :
STRUCT
	sObjectID					: STRING := 'MAIN.fbMMServer';
	sMethodID					: STRING := 'MAIN.fbMMServer#M_UpdateStationBuffer';
	iStatus						: INT;
	iNoOfInputArgs				: BYTE := 7;
	iNoOfOutputArgs				: BYTE := 2;
	stInput						: ST_UpdateStationBufferDataIn;
	stOutput					: ST_UpdateStationBufferDataOut;	
END_STRUCT
END_TYPE

// ---- ECC/Basic/TrackClient/Method Data/Data/ST_UpdateStationBufferDataIn.TcDUT
{attribute 'pack_mode' := '1'}
TYPE ST_UpdateStationBufferDataIn :
STRUCT
	sStationID					: STRING(30);								(* The ID of the station that will be moved to. *)
	eStationBufferType			: UINT; // E_MMStationBuffer;				(* Select pre or post buffer *)
	nIndex						: USINT;									(* Buffer index *)
	nVehicleID					: UINT;										(* Vehicle ID of vehicle at buffer position *)
	sCarrierID					: STRING(30);								(* Carrierr ID at buffer position *)
	nTicket						: UINT;										(* Ticket number *)
	nPriority					: UINT;										(* Ticket priority *)
END_STRUCT
END_TYPE

// ---- ECC/Basic/TrackClient/Method Data/Data/ST_UpdateStationBufferDataOut.TcDUT
{attribute 'pack_mode' := '1'}
TYPE ST_UpdateStationBufferDataOut :
STRUCT
	// Fixed data for all methods
	nNumberOfOutputArguments	: UDINT;								// determined amount of output parameters
	nReserved					: ARRAY[1..4] OF BYTE;					// Reserved padding
	
	// Method specific data
	stOutputArgInfo				: ARRAY[1..2] OF ST_UAMethodArgInfo; 	// 
	eStatus						: E_MMServerStatus;						// Status from remote method (succes/fail)
	sMessage					: STRING;								// Debugging message

END_STRUCT
END_TYPE

// ---- ECC/Basic/TrackClient/Method Data/Data/ST_UpdateVehicleDataData.TcDUT
TYPE ST_UpdateVehicleDataData :
STRUCT
	sObjectID					: STRING := 'MAIN.fbMMServer';
	sMethodID					: STRING := 'MAIN.fbMMServer#M_UpdateVehicleData';
	iStatus						: INT;
	iNoOfInputArgs				: BYTE := 10;
	iNoOfOutputArgs				: BYTE := 2;
	stInput						: ST_UpdateVehicleDataDataIn;
	stOutput					: ST_UpdateVehicleDataDataOut;	
END_STRUCT
END_TYPE

// ---- ECC/Basic/TrackClient/Method Data/Data/ST_UpdateVehicleDataDataIn.TcDUT
{attribute 'pack_mode' := '1'}
TYPE ST_UpdateVehicleDataDataIn :
STRUCT
	eInputType					: UINT;										(* The vehicle/vehicles that will be moved. *)
	sInput						: STRING(30);								(* Depending on the input type, the input can be the ID of a vehicle, last, article, last type, cell or station. *)
	sCarrierID					: STRING(30);								(* Carrier ID *)
	bTool						: BOOL;										(*  *)
	sToolID						: STRING(30);								(* Tool ID *)
	bMaterial					: BOOL;										(*  *)
	sMaterialID					: STRING(30);								(* Material ID string *)
	sJobID						: STRING(30);								(* Job ID string *)
	nTicket						: UINT;										(* Ticket number *)
	nPriority					: UINT;										(* Ticket priority *)
END_STRUCT
END_TYPE

// ---- ECC/Basic/TrackClient/Method Data/Data/ST_UpdateVehicleDataDataOut.TcDUT
{attribute 'pack_mode' := '1'}
TYPE ST_UpdateVehicleDataDataOut :
STRUCT
	// Fixed data for all methods
	nNumberOfOutputArguments	: UDINT;								// determined amount of output parameters
	nReserved					: ARRAY[1..4] OF BYTE;					// Reserved padding
	
	// Method specific data
	stOutputArgInfo				: ARRAY[1..2] OF ST_UAMethodArgInfo; 	// 
	eStatus						: E_MMServerStatus;						// Status from remote method (succes/fail)
	sMessage					: STRING;								// Debugging message

END_STRUCT
END_TYPE

// ---- ECC/Basic/TrackClient/Method Data/Data/ST_UpdateVehicleMappingDataData.TcDUT
TYPE ST_UpdateVehicleMappingDataData :
STRUCT
	sObjectID					: STRING := 'MAIN.fbMMServer';
	sMethodID					: STRING := 'MAIN.fbMMServer#M_UpdateVehicleMappingData';
	iStatus						: INT;
	iNoOfInputArgs				: BYTE := 6;
	iNoOfOutputArgs				: BYTE := 2;
	stInput						: ST_UpdateVehicleMappingDataDataIn;
	stOutput					: ST_UpdateVehicleMappingDataDataOut;	
END_STRUCT
END_TYPE

// ---- ECC/Basic/TrackClient/Method Data/Data/ST_UpdateVehicleMappingDataDataIn.TcDUT
{attribute 'pack_mode' := '1'}
TYPE ST_UpdateVehicleMappingDataDataIn :
STRUCT
	nVehicleID					: UINT;										(* Magnemotion vehicle ID *)
	sCarrierID					: STRING(30);								(* arrier ID (from RFID scan) *)
	bTool						: BOOL;										(* TRUE/FALSE (True if Tool mounted) *)
	sToolID						: STRING(30);								(* Tool ID (from RFID scan) *)
	bMaterial					: BOOL;										(* TRUE/FALSE (True if material in tray) *)
	sMaterialID					: STRING(30);								(* Material ID (from RFID Scan) (Optional) *)
END_STRUCT
END_TYPE

// ---- ECC/Basic/TrackClient/Method Data/Data/ST_UpdateVehicleMappingDataDataOut.TcDUT
{attribute 'pack_mode' := '1'}
TYPE ST_UpdateVehicleMappingDataDataOut :
STRUCT
	// Fixed data for all methods
	nNumberOfOutputArguments	: UDINT;								// determined amount of output parameters
	nReserved					: ARRAY[1..4] OF BYTE;					// Reserved padding
	
	// Method specific data
	stOutputArgInfo				: ARRAY[1..2] OF ST_UAMethodArgInfo; 	// 
	eStatus						: E_MMServerStatus;						// Status from remote method (succes/fail)
	sMessage					: STRING;								// Debugging message

END_STRUCT
END_TYPE

// ---- ECC/Basic/TrackClient/Method Data/Data/ST_UpdateVehicleMontageData.TcDUT
TYPE ST_UpdateVehicleMontageData :
STRUCT
	sObjectID					: STRING := 'MAIN.fbMMServer';
	sMethodID					: STRING := 'MAIN.fbMMServer#M_UpdateVehicleMontageData';
	iStatus						: INT;
	iNoOfInputArgs				: BYTE := 7;
	iNoOfOutputArgs				: BYTE := 2;
	stInput						: ST_UpdateVehicleMontageDataIn;
	stOutput					: ST_UpdateVehicleMontageDataOut;
END_STRUCT
END_TYPE

// ---- ECC/Basic/TrackClient/Method Data/Data/ST_UpdateVehicleMontageDataIn.TcDUT
{attribute 'pack_mode' := '1'}
TYPE ST_UpdateVehicleMontageDataIn :
STRUCT
	eInputType					: E_MMVehicleInputType;
	sInput						: STRING(30);										(* Identifier for the vehicle to update data for *)
	bTool						: BOOL;												(* TRUE if a tool is mounted *)
	sToolID						: STRING(30);										(* Tool ID for the mounted tool *)
	bMaterial					: BOOL;												(* TRUE if a material is mounted *)
	sMaterialID					: STRING(30);										(* Material ID for the mounted material *)
	bReserved					: BOOL;												(* TRUE if the vehicle should be reserved for montage loop *)
END_STRUCT
END_TYPE

// ---- ECC/Basic/TrackClient/Method Data/Data/ST_UpdateVehicleMontageDataOut.TcDUT
{attribute 'pack_mode' := '1'}
TYPE ST_UpdateVehicleMontageDataOut :
STRUCT
	// Fixed data for all methods
	nNumberOfOutputArguments	: UDINT;								// determined amount of output parameters
	nReserved					: ARRAY[1..4] OF BYTE;					// Reserved padding
	
	// Method specific data
	stOutputArgInfo				: ARRAY[1..2] OF ST_UAMethodArgInfo; 	// 
	eStatus						: E_MMServerStatus;						// Status from remote method (succes/fail)
	sMessage					: STRING;								// Debugging message

END_STRUCT
END_TYPE

// ---- ECC/Basic/TrackClient/Method Data/Data/ST_UpdateVehicleOwnerData.TcDUT
TYPE ST_UpdateVehicleOwnerData :
STRUCT
	sObjectID					: STRING := 'MAIN.fbMMServer';
	sMethodID					: STRING := 'MAIN.fbMMServer#M_UpdateVehicleOwner';
	iStatus						: INT;
	iNoOfInputArgs				: BYTE := 3;
	iNoOfOutputArgs				: BYTE := 2;
	stInput						: ST_UpdateVehicleOwnerDataIn;
	stOutput					: ST_UpdateVehicleOwnerDataOut;	
END_STRUCT
END_TYPE

// ---- ECC/Basic/TrackClient/Method Data/Data/ST_UpdateVehicleOwnerDataIn.TcDUT
{attribute 'pack_mode' := '1'}
TYPE ST_UpdateVehicleOwnerDataIn :
STRUCT
	eInputType					: UINT;										(* The vehicle/vehicles that will be moved. *)
	sInput						: STRING(30);								(* Depending on the input type, the input can be the ID of a vehicle, last, article, last type, cell or station. *)
	sCellID						: STRING(30);								(* Tool ID *)
END_STRUCT
END_TYPE

// ---- ECC/Basic/TrackClient/Method Data/Data/ST_UpdateVehicleOwnerDataOut.TcDUT
{attribute 'pack_mode' := '1'}
TYPE ST_UpdateVehicleOwnerDataOut :
STRUCT
	// Fixed data for all methods
	nNumberOfOutputArguments	: UDINT;								// determined amount of output parameters
	nReserved					: ARRAY[1..4] OF BYTE;					// Reserved padding
	
	// Method specific data
	stOutputArgInfo				: ARRAY[1..2] OF ST_UAMethodArgInfo; 	// 
	eStatus						: E_MMServerStatus;						// Status from remote method (succes/fail)
	sMessage					: STRING;								// Debugging message

END_STRUCT
END_TYPE

// ---- ECC/Basic/TrackClient/Method Data/Data/ST_UpdateVehicleReservationDataData.TcDUT
TYPE ST_UpdateVehicleReservationDataData :
STRUCT
	sObjectID					: STRING := 'MAIN.fbMMServer';
	sMethodID					: STRING := 'MAIN.fbMMServer#M_UpdateVehicleReservationData';
	iStatus						: INT;
	iNoOfInputArgs				: BYTE := 6;
	iNoOfOutputArgs				: BYTE := 2;
	stInput						: ST_UpdateVehicleReservationDataDataIn;
	stOutput					: ST_UpdateVehicleReservationDataDataOut;
END_STRUCT
END_TYPE

// ---- ECC/Basic/TrackClient/Method Data/Data/ST_UpdateVehicleReservationDataDataIn.TcDUT
{attribute 'pack_mode' := '1'}
TYPE ST_UpdateVehicleReservationDataDataIn :
STRUCT
	sTargetStationID			: STRING(30);										(* Station ID for the target station *)
	sCarrierID					: STRING(30);										(* Carrier ID (from RFID scan) *)
	sJobID						: STRING(30);										(* Job ID string *)
	nTicket						: UINT;												(* Ticket number *)
	nCarriersInPackage			: UINT;												(* Ticket Size *)
	nPriority					: UINT;												(* Ticket priority (within package) *)
END_STRUCT
END_TYPE

// ---- ECC/Basic/TrackClient/Method Data/Data/ST_UpdateVehicleReservationDataDataOut.TcDUT
{attribute 'pack_mode' := '1'}
TYPE ST_UpdateVehicleReservationDataDataOut :
STRUCT
	// Fixed data for all methods
	nNumberOfOutputArguments	: UDINT;								// determined amount of output parameters
	nReserved					: ARRAY[1..4] OF BYTE;					// Reserved padding
	
	// Method specific data
	stOutputArgInfo				: ARRAY[1..2] OF ST_UAMethodArgInfo; 	// 
	eStatus						: E_MMServerStatus;						// Status from remote method (succes/fail)
	sMessage					: STRING;								// Debugging message

END_STRUCT
END_TYPE

// ---- ECC/Basic/TrackClient/Method Data/Data/ST_UpdateVehicleReworkDataData.TcDUT
TYPE ST_UpdateVehicleReworkDataData :
STRUCT
	sObjectID					: STRING := 'MAIN.fbMMServer';
	sMethodID					: STRING := 'MAIN.fbMMServer#M_UpdateVehicleReworkData';
	iStatus						: INT;
	iNoOfInputArgs				: BYTE := 2;
	iNoOfOutputArgs				: BYTE := 2;
	stInput						: ST_UpdateVehicleReworkDataDataIn;
	stOutput					: ST_UpdateVehicleReworkDataDataOut;	
END_STRUCT
END_TYPE

// ---- ECC/Basic/TrackClient/Method Data/Data/ST_UpdateVehicleReworkDataDataIn.TcDUT
{attribute 'pack_mode' := '1'}
TYPE ST_UpdateVehicleReworkDataDataIn :
STRUCT
	sCarrierID					: STRING(30);								(* Carrier ID *)
	bNOK						: BOOL;										(* Rework required *)
END_STRUCT
END_TYPE

// ---- ECC/Basic/TrackClient/Method Data/Data/ST_UpdateVehicleReworkDataDataOut.TcDUT
{attribute 'pack_mode' := '1'}
TYPE ST_UpdateVehicleReworkDataDataOut :
STRUCT
	// Fixed data for all methods
	nNumberOfOutputArguments	: UDINT;								// determined amount of output parameters
	nReserved					: ARRAY[1..4] OF BYTE;					// Reserved padding
	
	// Method specific data
	stOutputArgInfo				: ARRAY[1..2] OF ST_UAMethodArgInfo; 	// 
	eStatus						: E_MMServerStatus;						// Status from remote method (succes/fail)
	sMessage					: STRING;								// Debugging message

END_STRUCT
END_TYPE

// ---- ECC/Basic/TrackClient/Method Data/MoveVehicle/ST_MoveToBufferData.TcDUT
TYPE ST_MoveToBufferData :
STRUCT
	sObjectID					: STRING := 'MAIN.fbMMServer';
	sMethodID					: STRING := 'MAIN.fbMMServer#M_MoveVehicleToStationBuffer2';
	iStatus						: INT;
	iNoOfInputArgs				: BYTE := 9;
	iNoOfOutputArgs				: BYTE := 3;
	stInput						: ST_MoveToBufferDataIn;
	stOutput					: ST_MoveToBufferDataOut;	
END_STRUCT
END_TYPE

// ---- ECC/Basic/TrackClient/Method Data/MoveVehicle/ST_MoveToBufferDataIn.TcDUT
{attribute 'pack_mode' := '1'}
TYPE ST_MoveToBufferDataIn :
STRUCT
	eInputType					: UINT;										(* The vehicle/vehicles that will be moved. *)
	sInput						: STRING(30);								(* Depending on the input type, the input can be the ID of a vehicle, last, article, last type, cell or station. *)
	sStationID					: STRING(30);								(* The ID of the station that will be moved to. *)
	eStationBufferType			: UINT; // E_MMStationBuffer;				(* Select pre or post buffer *)
	nIndex						: USINT;									(* Buffer index *)
	eDirection					: BYTE;										(* 0: BiDirectional, 1: Forward, 2: Backward *)
	nFollowID					: UINT := 0;
	fVelocity					: REAL;
	fAcceleration				: REAL;
END_STRUCT
END_TYPE

// ---- ECC/Basic/TrackClient/Method Data/MoveVehicle/ST_MoveToBufferDataOut.TcDUT
{attribute 'pack_mode' := '1'}
TYPE ST_MoveToBufferDataOut :
STRUCT
	// Fixed data for all methods
	nNumberOfOutputArguments	: UDINT;								// determined amount of output parameters
	nReserved					: ARRAY[1..4] OF BYTE;					// Reserved padding
	
	// Method specific data
	stOutputArgInfo				: ARRAY[1..3] OF ST_UAMethodArgInfo; 	// 
	eStatus						: E_MMServerStatus;						// Status from remote method (succes/fail)
	sMessage					: STRING;								// Debugging message
	iCommandID					: UINT;									// Command ID assigned by TrackServer to this command

END_STRUCT
END_TYPE

// ---- ECC/Basic/TrackClient/Method Data/MoveVehicle/ST_MoveToDecisionPointData.TcDUT
TYPE ST_MoveToDecisionPointData :
STRUCT
	sObjectID					: STRING := 'MAIN.fbMMServer';
	sMethodID					: STRING := 'MAIN.fbMMServer#M_MoveVehicleToStationDecisionPoint2';
	iStatus						: INT;
	iNoOfInputArgs				: BYTE := 7;
	iNoOfOutputArgs				: BYTE := 3;
	stInput						: ST_MoveToDecisionPointDataIn;
	stOutput					: ST_MoveToDecisionPointDataOut;	
END_STRUCT
END_TYPE

// ---- ECC/Basic/TrackClient/Method Data/MoveVehicle/ST_MoveToDecisionPointDataIn.TcDUT
{attribute 'pack_mode' := '1'}
TYPE ST_MoveToDecisionPointDataIn :
STRUCT
	eInputType					: UINT;										(* The vehicle/vehicles that will be moved. *)
	sInput						: STRING(30);									(* Depending on the input type, the input can be the ID of a vehicle, last, article, last type, cell or station. *)
	sStationID					: STRING(30);									(* The ID of the station that will be moved to. *)
	eDirection					: BYTE;										(* 0: BiDirectional, 1: Forward, 2: Backward *)
	nFollowID					: UINT := 0;
	fVelocity					: REAL;
	fAcceleration				: REAL;
END_STRUCT
END_TYPE

// ---- ECC/Basic/TrackClient/Method Data/MoveVehicle/ST_MoveToDecisionPointDataOut.TcDUT
{attribute 'pack_mode' := '1'}
TYPE ST_MoveToDecisionPointDataOut :
STRUCT
	// Fixed data for all methods
	nNumberOfOutputArguments	: UDINT;								// determined amount of output parameters
	nReserved					: ARRAY[1..4] OF BYTE;					// Reserved padding
	
	// Method specific data
	stOutputArgInfo				: ARRAY[1..3] OF ST_UAMethodArgInfo; 	// 
	eStatus						: E_MMServerStatus;						// Status from remote method (succes/fail)
	sMessage					: STRING;								// Debugging message	
	iCommandID					: UINT;									// Command ID assigned by TrackServer to this command

END_STRUCT
END_TYPE

// ---- ECC/Basic/TrackClient/Method Data/MoveVehicle/ST_MoveToPositionData.TcDUT
TYPE ST_MoveToPositionData :
STRUCT
	sObjectID					: STRING := 'MAIN.fbMMServer';
	sMethodID					: STRING := 'MAIN.fbMMServer#M_MoveVehicleToPosition2';
	iStatus						: INT;
	iNoOfInputArgs				: BYTE := 8;
	iNoOfOutputArgs				: BYTE := 3;
	stInput						: ST_MoveToPositionDataIn;
	stOutput					: ST_MoveToPositionDataOut;	
END_STRUCT
END_TYPE

// ---- ECC/Basic/TrackClient/Method Data/MoveVehicle/ST_MoveToPositionDataIn.TcDUT
{attribute 'pack_mode' := '1'}
TYPE ST_MoveToPositionDataIn :
STRUCT
	eInputType					: UINT;										(* The vehicle/vehicles that will be moved. *)
	sInput						: STRING(30);								(* Depending on the input type, the input can be the ID of a vehicle, last, article, last type, cell or station. *)
	nPathID						: UINT;										(* The ID of the target Path *)
	fPosition					: REAL;										(* The position on the speciied Path *)
	eDirection					: BYTE;										(* 0: BiDirectional, 1: Forward, 2: Backward *)
	nFollowID					: UINT := 0;
	fVelocity					: REAL;
	fAcceleration				: REAL;
END_STRUCT
END_TYPE

// ---- ECC/Basic/TrackClient/Method Data/MoveVehicle/ST_MoveToPositionDataOut.TcDUT
{attribute 'pack_mode' := '1'}
TYPE ST_MoveToPositionDataOut :
STRUCT
	// Fixed data for all methods
	nNumberOfOutputArguments	: UDINT;								// determined amount of output parameters
	nReserved					: ARRAY[1..4] OF BYTE;					// Reserved padding
	
	// Method specific data
	stOutputArgInfo				: ARRAY[1..3] OF ST_UAMethodArgInfo; 	// 
	eStatus						: E_MMServerStatus;						// Status from remote method (succes/fail)
	sMessage					: STRING;								// Debugging message
	iCommandID					: UINT;									// Command ID assigned by TrackServer to this command

END_STRUCT
END_TYPE

// ---- ECC/Basic/TrackClient/Method Data/MoveVehicle/ST_MoveToScannerData.TcDUT
TYPE ST_MoveToScannerData :
STRUCT
	sObjectID					: STRING := 'MAIN.fbMMServer';
	sMethodID					: STRING := 'MAIN.fbMMServer#M_MoveVehicleToScanner2';
	iStatus						: INT;
	iNoOfInputArgs				: BYTE := 4;
	iNoOfOutputArgs				: BYTE := 3;
	stInput						: ST_MoveToScannerDataIn;
	stOutput					: ST_MoveToScannerDataOut;	
END_STRUCT
END_TYPE

// ---- ECC/Basic/TrackClient/Method Data/MoveVehicle/ST_MoveToScannerDataIn.TcDUT
{attribute 'pack_mode' := '1'}
TYPE ST_MoveToScannerDataIn :
STRUCT
	eInputType					: UINT;										(* The vehicle/vehicles that will be moved. *)
	sInput						: STRING(30);								(* Depending on the input type, the input can be the ID of a vehicle, last, article, last type, cell or station. *)
	eDirection					: BYTE;										(* 0: BiDirectional, 1: Forward, 2: Backward *)
	nFollowID					: UINT := 0;
	fVelocity					: REAL;
	fAcceleration				: REAL;
END_STRUCT
END_TYPE

// ---- ECC/Basic/TrackClient/Method Data/MoveVehicle/ST_MoveToScannerDataOut.TcDUT
{attribute 'pack_mode' := '1'}
TYPE ST_MoveToScannerDataOut :
STRUCT
	// Fixed data for all methods
	nNumberOfOutputArguments	: UDINT;								// determined amount of output parameters
	nReserved					: ARRAY[1..4] OF BYTE;					// Reserved padding
	
	// Method specific data
	stOutputArgInfo				: ARRAY[1..3] OF ST_UAMethodArgInfo; 	// 
	eStatus						: E_MMServerStatus;						// Status from remote method (succes/fail)
	sMessage					: STRING;								// Debugging message
	iCommandID					: UINT;									// Command ID assigned by TrackServer to this command

END_STRUCT
END_TYPE

// ---- ECC/Basic/TrackClient/Method Data/MoveVehicle/ST_MoveToStationDataIn.TcDUT
{attribute 'pack_mode' := '1'}
TYPE ST_MoveToStationDataIn :
STRUCT
	eInputType					: UINT;										(* The vehicle/vehicles that will be moved. *)
	sInput						: STRING(30);								(* Depending on the input type, the input can be the ID of a vehicle, last, article, last type, cell or station. *)
	sStationID					: STRING(30);								(* The ID of the station that will be moved to. *)
	eDirection					: BYTE;										(* 0: BiDirectional, 1: Forward, 2: Backward *)
	nFollowID					: UINT := 0;
	fVelocity					: REAL;
	fAcceleration				: REAL;
END_STRUCT
END_TYPE

// ---- ECC/Basic/TrackClient/Method Data/MoveVehicle/ST_MoveToStationDataOut.TcDUT
{attribute 'pack_mode' := '1'}
TYPE ST_MoveToStationDataOut :
STRUCT
	// Fixed data for all methods
	nNumberOfOutputArguments	: UDINT;								// determined amount of output parameters
	nReserved					: ARRAY[1..4] OF BYTE;					// Reserved padding
	
	// Method specific data
	stOutputArgInfo				: ARRAY[1..3] OF ST_UAMethodArgInfo; 	// 
	eStatus						: E_MMServerStatus;						// Status from remote method (succes/fail)
	sMessage					: STRING;								// Debugging message
	iCommandID					: UINT;									// Command ID assigned by TrackServer to this command

END_STRUCT
END_TYPE

// ---- ECC/Basic/TrackClient/Method Data/MoveVehicle/ST_MoveToStationInData.TcDUT
TYPE ST_MoveToStationInData :
STRUCT
	sObjectID					: STRING := 'MAIN.fbMMServer';
	sMethodID					: STRING := 'MAIN.fbMMServer#M_MoveVehicleToStationIn2';
	iStatus						: INT;
	iNoOfInputArgs				: BYTE := 7;
	iNoOfOutputArgs				: BYTE := 3;
	stInput						: ST_MoveToStationDataIn;
	stOutput					: ST_MoveToStationDataOut;	
END_STRUCT
END_TYPE

// ---- ECC/Basic/TrackClient/Method Data/MoveVehicle/ST_MoveToStationOutData.TcDUT
TYPE ST_MoveToStationOutData :
STRUCT
	sObjectID					: STRING := 'MAIN.fbMMServer';
	sMethodID					: STRING := 'MAIN.fbMMServer#M_MoveVehicleToStationOut2';
	iStatus						: INT;
	iNoOfInputArgs				: BYTE := 7;
	iNoOfOutputArgs				: BYTE := 3;
	stInput						: ST_MoveToStationDataIn;
	stOutput					: ST_MoveToStationDataOut;	
END_STRUCT
END_TYPE

// ---- ECC/Basic/TrackClient/Method Data/MoveVehicle/ST_MoveVehicleStatusData.TcDUT
TYPE ST_MoveVehicleStatusData :
STRUCT
	sObjectID					: STRING := 'MAIN.fbMMServer';
	sMethodID					: STRING := 'MAIN.fbMMServer#M_MoveVehicleStatus';
	iStatus						: INT;
	iNoOfInputArgs				: BYTE := 1;
	iNoOfOutputArgs				: BYTE := 3;
	stInput						: ST_MoveVehicleStatusDataIn;
	stOutput					: ST_MoveVehicleStatusDataOut;	
END_STRUCT
END_TYPE

// ---- ECC/Basic/TrackClient/Method Data/MoveVehicle/ST_MoveVehicleStatusDataIn.TcDUT
{attribute 'pack_mode' := '1'}
TYPE ST_MoveVehicleStatusDataIn :
STRUCT
	iCommandID					: UINT;													// The command ID for this command

END_STRUCT
END_TYPE

// ---- ECC/Basic/TrackClient/Method Data/MoveVehicle/ST_MoveVehicleStatusDataOut.TcDUT
{attribute 'pack_mode' := '1'}
TYPE ST_MoveVehicleStatusDataOut :
STRUCT
	// Fixed data for all methods
	nNumberOfOutputArguments	: UDINT;								// determined amount of output parameters
	nReserved					: ARRAY[1..4] OF BYTE;					// Reserved padding
	
	// Method specific data
	stOutputArgInfo				: ARRAY[1..3] OF ST_UAMethodArgInfo; 	// 
	eStatus						: E_MMServerStatus;						// Status from remote method (succes/fail)
	sMessage					: STRING;								// Debugging message	
	eMoveStatus					: E_VehicleMoveState;					// Status of movement

END_STRUCT
END_TYPE

// ---- ECC/Basic/TrackClient/Method Data/Path/ST_AddPathData.TcDUT
TYPE ST_AddPathData :
STRUCT
	sObjectID					: STRING := 'MAIN.fbMMServer';
	sMethodID					: STRING := 'MAIN.fbMMServer#M_AddPath';
	iStatus						: INT;
	iNoOfInputArgs				: BYTE := 3;
	iNoOfOutputArgs				: BYTE := 2;
	stInput						: ST_AddPathDataIn;
	stOutput					: ST_AddPathDataOut;	
END_STRUCT
END_TYPE

// ---- ECC/Basic/TrackClient/Method Data/Path/ST_AddPathDataIn.TcDUT
{attribute 'pack_mode' := '1'}
TYPE ST_AddPathDataIn :
STRUCT
	sCellID						: STRING(30);	// 
	iPath						: UINT;			// MM path ID (1-65536)
	bPresent					: BOOL;			// 
END_STRUCT
END_TYPE

// ---- ECC/Basic/TrackClient/Method Data/Path/ST_AddPathDataOut.TcDUT
{attribute 'pack_mode' := '1'}
TYPE ST_AddPathDataOut :
STRUCT
	// Fixed data for all methods
	nNumberOfOutputArguments	: UDINT;								// determined amount of output parameters
	nReserved					: ARRAY[1..4] OF BYTE;					// Reserved padding
	
	// Method specific data
	stOutputArgInfo				: ARRAY[1..2] OF ST_UAMethodArgInfo; 	// 
	eStatus						: E_MMServerStatus;						// Status from remote method (succes/fail)
	sMessage					: STRING;								// Debugging message

END_STRUCT
END_TYPE

// ---- ECC/Basic/TrackClient/Method Data/Path/ST_RemovePathData.TcDUT
TYPE ST_RemovePathData :
STRUCT
	sObjectID					: STRING := 'MAIN.fbMMServer';
	sMethodID					: STRING := 'MAIN.fbMMServer#M_RemovePath';
	iStatus						: INT;
	iNoOfInputArgs				: BYTE := 2;
	iNoOfOutputArgs				: BYTE := 2;
	stInput						: ST_RemovePathDataIn;
	stOutput					: ST_RemovePathDataOut;	
END_STRUCT
END_TYPE

// ---- ECC/Basic/TrackClient/Method Data/Path/ST_RemovePathDataIn.TcDUT
{attribute 'pack_mode' := '1'}
TYPE ST_RemovePathDataIn :
STRUCT
	sCellID						: STRING(30);	// 
	iPath						: UINT;			// MM path ID (1-65536)
END_STRUCT
END_TYPE

// ---- ECC/Basic/TrackClient/Method Data/Path/ST_RemovePathDataOut.TcDUT
{attribute 'pack_mode' := '1'}
TYPE ST_RemovePathDataOut :
STRUCT
	// Fixed data for all methods
	nNumberOfOutputArguments	: UDINT;								// determined amount of output parameters
	nReserved					: ARRAY[1..4] OF BYTE;					// Reserved padding
	
	// Method specific data
	stOutputArgInfo				: ARRAY[1..2] OF ST_UAMethodArgInfo; 	// 
	eStatus						: E_MMServerStatus;						// Status from remote method (succes/fail)
	sMessage					: STRING;								// Debugging message

END_STRUCT
END_TYPE

// ---- ECC/Basic/TrackClient/Method Data/Path/ST_ResetPathData.TcDUT
TYPE ST_ResetPathData :
STRUCT
	sObjectID					: STRING := 'MAIN.fbMMServer';
	sMethodID					: STRING := 'MAIN.fbMMServer#M_ResetPath';
	iStatus						: INT;
	iNoOfInputArgs				: BYTE := 1;
	iNoOfOutputArgs				: BYTE := 2;
	stInput						: ST_ResetPathDataIn;
	stOutput					: ST_ResetPathDataOut;	
END_STRUCT
END_TYPE

// ---- ECC/Basic/TrackClient/Method Data/Path/ST_ResetPathDataIn.TcDUT
{attribute 'pack_mode' := '1'}
TYPE ST_ResetPathDataIn :
STRUCT
	iPath						: UINT;			// MM path ID (1-65536)
END_STRUCT
END_TYPE

// ---- ECC/Basic/TrackClient/Method Data/Path/ST_ResetPathDataOut.TcDUT
{attribute 'pack_mode' := '1'}
TYPE ST_ResetPathDataOut :
STRUCT
	// Fixed data for all methods
	nNumberOfOutputArguments	: UDINT;								// determined amount of output parameters
	nReserved					: ARRAY[1..4] OF BYTE;					// Reserved padding
	
	// Method specific data
	stOutputArgInfo				: ARRAY[1..2] OF ST_UAMethodArgInfo; 	// 
	eStatus						: E_MMServerStatus;						// Status from remote method (succes/fail)
	sMessage					: STRING;								// Debugging message

END_STRUCT
END_TYPE

// ---- ECC/Basic/TrackClient/Method Data/Path/ST_ResumePathData.TcDUT
TYPE ST_ResumePathData :
STRUCT
	sObjectID					: STRING := 'MAIN.fbMMServer';
	sMethodID					: STRING := 'MAIN.fbMMServer#M_ResumePath';
	iStatus						: INT;
	iNoOfInputArgs				: BYTE := 1;
	iNoOfOutputArgs				: BYTE := 2;
	stInput						: ST_ResumePathDataIn;
	stOutput					: ST_ResumePathDataOut;	
END_STRUCT
END_TYPE

// ---- ECC/Basic/TrackClient/Method Data/Path/ST_ResumePathDataIn.TcDUT
{attribute 'pack_mode' := '1'}
TYPE ST_ResumePathDataIn :
STRUCT
	iPath						: UINT;			// MM path ID (1-65536)
END_STRUCT
END_TYPE

// ---- ECC/Basic/TrackClient/Method Data/Path/ST_ResumePathDataOut.TcDUT
{attribute 'pack_mode' := '1'}
TYPE ST_ResumePathDataOut :
STRUCT
	// Fixed data for all methods
	nNumberOfOutputArguments	: UDINT;								// determined amount of output parameters
	nReserved					: ARRAY[1..4] OF BYTE;					// Reserved padding
	
	// Method specific data
	stOutputArgInfo				: ARRAY[1..2] OF ST_UAMethodArgInfo; 	// 
	eStatus						: E_MMServerStatus;						// Status from remote method (succes/fail)
	sMessage					: STRING;								// Debugging message

END_STRUCT
END_TYPE

// ---- ECC/Basic/TrackClient/Method Data/Path/ST_StartPathData.TcDUT
TYPE ST_StartPathData :
STRUCT
	sObjectID					: STRING := 'MAIN.fbMMServer';
	sMethodID					: STRING := 'MAIN.fbMMServer#M_StartPath';
	iStatus						: INT;
	iNoOfInputArgs				: BYTE := 1;
	iNoOfOutputArgs				: BYTE := 2;
	stInput						: ST_StartPathDataIn;
	stOutput					: ST_StartPathDataOut;	
END_STRUCT
END_TYPE

// ---- ECC/Basic/TrackClient/Method Data/Path/ST_StartPathDataIn.TcDUT
{attribute 'pack_mode' := '1'}
TYPE ST_StartPathDataIn :
STRUCT
	iPath						: UINT;			// MM path ID (1-65536)
END_STRUCT
END_TYPE

// ---- ECC/Basic/TrackClient/Method Data/Path/ST_StartPathDataOut.TcDUT
{attribute 'pack_mode' := '1'}
TYPE ST_StartPathDataOut :
STRUCT
	// Fixed data for all methods
	nNumberOfOutputArguments	: UDINT;								// determined amount of output parameters
	nReserved					: ARRAY[1..4] OF BYTE;					// Reserved padding
	
	// Method specific data
	stOutputArgInfo				: ARRAY[1..2] OF ST_UAMethodArgInfo; 	// 
	eStatus						: E_MMServerStatus;						// Status from remote method (succes/fail)
	sMessage					: STRING;								// Debugging message

END_STRUCT
END_TYPE

// ---- ECC/Basic/TrackClient/Method Data/Path/ST_SuspendPathData.TcDUT
TYPE ST_SuspendPathData :
STRUCT
	sObjectID					: STRING := 'MAIN.fbMMServer';
	sMethodID					: STRING := 'MAIN.fbMMServer#M_SuspendPath';
	iStatus						: INT;
	iNoOfInputArgs				: BYTE := 1;
	iNoOfOutputArgs				: BYTE := 2;
	stInput						: ST_SuspendPathDataIn;
	stOutput					: ST_SuspendPathDataOut;	
END_STRUCT
END_TYPE

// ---- ECC/Basic/TrackClient/Method Data/Path/ST_SuspendPathDataIn.TcDUT
{attribute 'pack_mode' := '1'}
TYPE ST_SuspendPathDataIn :
STRUCT
	iPath						: UINT;			// MM path ID (1-65536)
END_STRUCT
END_TYPE

// ---- ECC/Basic/TrackClient/Method Data/Path/ST_SuspendPathDataOut.TcDUT
{attribute 'pack_mode' := '1'}
TYPE ST_SuspendPathDataOut :
STRUCT
	// Fixed data for all methods
	nNumberOfOutputArguments	: UDINT;								// determined amount of output parameters
	nReserved					: ARRAY[1..4] OF BYTE;					// Reserved padding
	
	// Method specific data
	stOutputArgInfo				: ARRAY[1..2] OF ST_UAMethodArgInfo; 	// 
	eStatus						: E_MMServerStatus;						// Status from remote method (succes/fail)
	sMessage					: STRING;								// Debugging message

END_STRUCT
END_TYPE

// ---- ECC/Basic/TrackClient/Method Data/Segment/ST_AddPathSegmentData.TcDUT
TYPE ST_AddPathSegmentData :
STRUCT
	sObjectID					: STRING := 'MAIN.fbMMServer';
	sMethodID					: STRING := 'MAIN.fbMMServer#M_AddPathSegment';
	iStatus						: INT;
	iNoOfInputArgs				: BYTE := 5;
	iNoOfOutputArgs				: BYTE := 2;
	stInput						: ST_AddPathSegmentDataIn;
	stOutput					: ST_AddPathSegmentDataOut;	
END_STRUCT
END_TYPE

// ---- ECC/Basic/TrackClient/Method Data/Segment/ST_AddPathSegmentDataIn.TcDUT
{attribute 'pack_mode' := '1'}
TYPE ST_AddPathSegmentDataIn :
STRUCT
	sCellID						: STRING(30);	// 
	sSegmentID					: STRING(30);	// 
	iPath						: UINT;			// MM path ID (1-65536)
	rBeginPosition				: REAL;			// The position of the start of the segment
	rEndPosition				: REAL;			// The position of the end of the segment (If position is greater than physical end
												// position, the segment will cover until the end of the path!)
END_STRUCT
END_TYPE

// ---- ECC/Basic/TrackClient/Method Data/Segment/ST_AddPathSegmentDataOut.TcDUT
{attribute 'pack_mode' := '1'}
TYPE ST_AddPathSegmentDataOut :
STRUCT
	// Fixed data for all methods
	nNumberOfOutputArguments	: UDINT;								// determined amount of output parameters
	nReserved					: ARRAY[1..4] OF BYTE;					// Reserved padding
	
	// Method specific data
	stOutputArgInfo				: ARRAY[1..2] OF ST_UAMethodArgInfo; 	// 
	eStatus						: E_MMServerStatus;						// Status from remote method (succes/fail)
	sMessage					: STRING;								// Debugging message

END_STRUCT
END_TYPE

// ---- ECC/Basic/TrackClient/Method Data/Segment/ST_GetPathSegmentVehicleCountData.TcDUT
TYPE ST_GetPathSegmentVehicleCountData :
STRUCT
	sObjectID					: STRING := 'MAIN.fbMMServer';
	sMethodID					: STRING := 'MAIN.fbMMServer#M_GetPathSegmentVehicleCount';
	iStatus						: INT;
	iNoOfInputArgs				: BYTE := 2;
	iNoOfOutputArgs				: BYTE := 3;
	stInput						: ST_GetPathSegmentVehicleCountDataIn;
	stOutput					: ST_GetPathSegmentVehicleCountDataOut;	
END_STRUCT
END_TYPE

// ---- ECC/Basic/TrackClient/Method Data/Segment/ST_GetPathSegmentVehicleCountDataIn.TcDUT
{attribute 'pack_mode' := '1'}
TYPE ST_GetPathSegmentVehicleCountDataIn :
STRUCT
	sCellID						: STRING(30);	// 
	sSegmentID					: STRING(30);	// 

END_STRUCT
END_TYPE

// ---- ECC/Basic/TrackClient/Method Data/Segment/ST_GetPathSegmentVehicleCountDataOut.TcDUT
{attribute 'pack_mode' := '1'}
TYPE ST_GetPathSegmentVehicleCountDataOut :
STRUCT
	// Fixed data for all methods
	nNumberOfOutputArguments	: UDINT;								// determined amount of output parameters
	nReserved					: ARRAY[1..4] OF BYTE;					// Reserved padding
	
	// Method specific data
	stOutputArgInfo				: ARRAY[1..3] OF ST_UAMethodArgInfo; 	// 
	iVehicleCount				: UINT;									// Number of vehicles on the segment
	eStatus						: E_MMServerStatus;						// Status from remote method (succes/fail)
	sMessage					: STRING;								// Debugging message

END_STRUCT
END_TYPE

// ---- ECC/Basic/TrackClient/Method Data/Segment/ST_RemovePathSegmentData.TcDUT
TYPE ST_RemovePathSegmentData :
STRUCT
	sObjectID					: STRING := 'MAIN.fbMMServer';
	sMethodID					: STRING := 'MAIN.fbMMServer#M_RemovePathSegment';
	iStatus						: INT;
	iNoOfInputArgs				: BYTE := 2;
	iNoOfOutputArgs				: BYTE := 2;
	stInput						: ST_RemovePathSegmentDataIn;
	stOutput					: ST_RemovePathSegmentDataOut;	
END_STRUCT
END_TYPE

// ---- ECC/Basic/TrackClient/Method Data/Segment/ST_RemovePathSegmentDataIn.TcDUT
{attribute 'pack_mode' := '1'}
TYPE ST_RemovePathSegmentDataIn :
STRUCT
	sCellID						: STRING(30);	// 
	sSegmentID					: STRING(30);	// 
												// position, the segment will cover until the end of the path!)
END_STRUCT
END_TYPE

// ---- ECC/Basic/TrackClient/Method Data/Segment/ST_RemovePathSegmentDataOut.TcDUT
{attribute 'pack_mode' := '1'}
TYPE ST_RemovePathSegmentDataOut :
STRUCT
	// Fixed data for all methods
	nNumberOfOutputArguments	: UDINT;								// determined amount of output parameters
	nReserved					: ARRAY[1..4] OF BYTE;					// Reserved padding
	
	// Method specific data
	stOutputArgInfo				: ARRAY[1..2] OF ST_UAMethodArgInfo; 	// 
	eStatus						: E_MMServerStatus;						// Status from remote method (succes/fail)
	sMessage					: STRING;								// Debugging message

END_STRUCT
END_TYPE

// ---- ECC/Basic/TrackClient/Method Data/Station/ST_AddStationData.TcDUT
TYPE ST_AddStationData :
STRUCT
	sObjectID					: STRING := 'MAIN.fbMMServer';
	sMethodID					: STRING := 'MAIN.fbMMServer#M_AddStation';
	iStatus						: INT;
	iNoOfInputArgs				: BYTE := 10;
	iNoOfOutputArgs				: BYTE := 2;
	stInput						: ST_AddStationDataIn;
	stOutput					: ST_AddStationDataOut;	
END_STRUCT
END_TYPE

// ---- ECC/Basic/TrackClient/Method Data/Station/ST_AddStationDataIn.TcDUT
{attribute 'pack_mode' := '1'}
TYPE ST_AddStationDataIn :
STRUCT
	sCellID						: STRING(30);
	sID							: STRING(30);
	iInPath						: UINT;
	rInPosition					: REAL;
	iOutPath					: UINT;
	rOutPosition				: REAL;
	iDecisionPath				: UINT;
	rDecisionPosition			: REAL;
	nPreBufferSize				: UINT;
	nPostBufferSize				: UINT;
END_STRUCT
END_TYPE

// ---- ECC/Basic/TrackClient/Method Data/Station/ST_AddStationDataOut.TcDUT
{attribute 'pack_mode' := '1'}
TYPE ST_AddStationDataOut :
STRUCT
	// Fixed data for all methods
	nNumberOfOutputArguments	: UDINT;								// determined amount of output parameters
	nReserved					: ARRAY[1..4] OF BYTE;					// Reserved padding
	
	// Method specific data
	stOutputArgInfo				: ARRAY[1..2] OF ST_UAMethodArgInfo; 	// 
	eStatus						: E_MMServerStatus;						// Status from remote method (succes/fail)
	sMessage					: STRING;								// Debugging message

END_STRUCT
END_TYPE

// ---- ECC/Basic/TrackClient/Method Data/Station/ST_AddStationDoubleData.TcDUT
TYPE ST_AddStationDoubleData :
STRUCT
	sObjectID					: STRING := 'MAIN.fbMMServer';
	sMethodID					: STRING := 'MAIN.fbMMServer#M_AddStationDouble';
	iStatus						: INT;
	iNoOfInputArgs				: BYTE := 10;
	iNoOfOutputArgs				: BYTE := 2;
	stInput						: ST_AddStationDoubleDataIn;
	stOutput					: ST_AddStationDoubleDataOut;	
END_STRUCT
END_TYPE

// ---- ECC/Basic/TrackClient/Method Data/Station/ST_AddStationDoubleDataIn.TcDUT
{attribute 'pack_mode' := '1'}
TYPE ST_AddStationDoubleDataIn :
STRUCT
	sCellID						: STRING(30);
	sID							: STRING(30);
	iInPath						: UINT;
	rInPosition					: REAL;
	iOutPath					: UINT;
	rOutPosition				: REAL;
	iDecisionPath				: UINT;
	rDecisionPosition			: REAL;
	nPreBufferSize				: UINT;
	nPostBufferSize				: UINT;
END_STRUCT
END_TYPE

// ---- ECC/Basic/TrackClient/Method Data/Station/ST_AddStationDoubleDataOut.TcDUT
{attribute 'pack_mode' := '1'}
TYPE ST_AddStationDoubleDataOut :
STRUCT
	// Fixed data for all methods
	nNumberOfOutputArguments	: UDINT;								// determined amount of output parameters
	nReserved					: ARRAY[1..4] OF BYTE;					// Reserved padding
	
	// Method specific data
	stOutputArgInfo				: ARRAY[1..2] OF ST_UAMethodArgInfo; 	// 
	eStatus						: E_MMServerStatus;						// Status from remote method (succes/fail)
	sMessage					: STRING;								// Debugging message

END_STRUCT
END_TYPE

// ---- ECC/Basic/TrackClient/Method Data/Station/ST_AddStationSingleData.TcDUT
TYPE ST_AddStationSingleData :
STRUCT
	sObjectID					: STRING := 'MAIN.fbMMServer';
	sMethodID					: STRING := 'MAIN.fbMMServer#M_AddStationSingle';
	iStatus						: INT;
	iNoOfInputArgs				: BYTE := 8;
	iNoOfOutputArgs				: BYTE := 2;
	stInput						: ST_AddStationSingleDataIn;
	stOutput					: ST_AddStationSingleDataOut;	
END_STRUCT
END_TYPE

// ---- ECC/Basic/TrackClient/Method Data/Station/ST_AddStationSingleDataIn.TcDUT
{attribute 'pack_mode' := '1'}
TYPE ST_AddStationSingleDataIn :
STRUCT
	sCellID						: STRING(30);
	sID							: STRING(30);
	iPath						: UINT;
	rPosition					: REAL;
	iDecisionPath				: UINT;
	rDecisionPosition			: REAL;
	nPreBufferSize				: UINT;
	nPostBufferSize				: UINT;
END_STRUCT
END_TYPE

// ---- ECC/Basic/TrackClient/Method Data/Station/ST_AddStationSingleDataOut.TcDUT
{attribute 'pack_mode' := '1'}
TYPE ST_AddStationSingleDataOut :
STRUCT
	// Fixed data for all methods
	nNumberOfOutputArguments	: UDINT;								// determined amount of output parameters
	nReserved					: ARRAY[1..4] OF BYTE;					// Reserved padding
	
	// Method specific data
	stOutputArgInfo				: ARRAY[1..2] OF ST_UAMethodArgInfo; 	// 
	eStatus						: E_MMServerStatus;						// Status from remote method (succes/fail)
	sMessage					: STRING;								// Debugging message

END_STRUCT
END_TYPE

// ---- ECC/Basic/TrackClient/Method Data/Station/ST_AdjustBufferPosData.TcDUT
TYPE ST_AdjustBufferPosData :
STRUCT
	sObjectID					: STRING := 'MAIN.fbMMServer';
	sMethodID					: STRING := 'MAIN.fbMMServer#M_AdjustBufferPosition';
	iStatus						: INT;
	iNoOfInputArgs				: BYTE := 3;
	iNoOfOutputArgs				: BYTE := 2;
	stInput						: ST_AdjustBufferPosDataIn;
	stOutput					: ST_AdjustBufferPosDataOut;	
END_STRUCT
END_TYPE

// ---- ECC/Basic/TrackClient/Method Data/Station/ST_AdjustBufferPosDataIn.TcDUT
{attribute 'pack_mode' := '1'}
TYPE ST_AdjustBufferPosDataIn :
STRUCT
	sStationID			: STRING;				// Station ID (e.g. S00000A)
	eBufferType			: E_MMStationBuffer;	// Pre- or Post-buffer
	rDistance			: REAL;					// [M] Distance in metres (negative value to move backwards)
END_STRUCT
END_TYPE

// ---- ECC/Basic/TrackClient/Method Data/Station/ST_AdjustBufferPosDataOut.TcDUT
{attribute 'pack_mode' := '1'}
TYPE ST_AdjustBufferPosDataOut :
STRUCT
	// Fixed data for all methods
	nNumberOfOutputArguments	: UDINT;								// determined amount of output parameters
	nReserved					: ARRAY[1..4] OF BYTE;					// Reserved padding
	
	// Method specific data
	stOutputArgInfo				: ARRAY[1..2] OF ST_UAMethodArgInfo; 	// 
	eStatus						: E_MMServerStatus;						// Status from remote method (succes/fail)
	sMessage					: STRING;								// Debugging message

END_STRUCT
END_TYPE

// ---- ECC/Basic/TrackClient/Method Data/Station/ST_EnableStationData.TcDUT
TYPE ST_EnableStationData :
STRUCT
	sObjectID					: STRING := 'MAIN.fbMMServer';
	sMethodID					: STRING := 'MAIN.fbMMServer#M_AddStation2';
	iStatus						: INT;
	iNoOfInputArgs				: BYTE := 3;
	iNoOfOutputArgs				: BYTE := 2;
	stInput						: ST_EnableStationDataIn;
	stOutput					: ST_EnableStationDataOut;	
END_STRUCT
END_TYPE

// ---- ECC/Basic/TrackClient/Method Data/Station/ST_EnableStationDataIn.TcDUT
{attribute 'pack_mode' := '1'}
TYPE ST_EnableStationDataIn :
STRUCT
	sCellID						: STRING(30);
	sID							: STRING(30);
	bPresent					: BOOL;
END_STRUCT
END_TYPE

// ---- ECC/Basic/TrackClient/Method Data/Station/ST_EnableStationDataOut.TcDUT
{attribute 'pack_mode' := '1'}
TYPE ST_EnableStationDataOut :
STRUCT
	// Fixed data for all methods
	nNumberOfOutputArguments	: UDINT;								// determined amount of output parameters
	nReserved					: ARRAY[1..4] OF BYTE;					// Reserved padding
	
	// Method specific data
	stOutputArgInfo				: ARRAY[1..2] OF ST_UAMethodArgInfo; 	// 
	eStatus						: E_MMServerStatus;						// Status from remote method (succes/fail)
	sMessage					: STRING;								// Debugging message

END_STRUCT
END_TYPE

// ---- ECC/Basic/TrackClient/Method Data/Station/ST_RemoveStationData.TcDUT
TYPE ST_RemoveStationData :
STRUCT
	sObjectID					: STRING := 'MAIN.fbMMServer';
	sMethodID					: STRING := 'MAIN.fbMMServer#M_RemoveStation';
	iStatus						: INT;
	iNoOfInputArgs				: BYTE := 2;
	iNoOfOutputArgs				: BYTE := 2;
	stInput						: ST_RemoveStationDataIn;
	stOutput					: ST_RemoveStationDataOut;	
END_STRUCT
END_TYPE

// ---- ECC/Basic/TrackClient/Method Data/Station/ST_RemoveStationDataIn.TcDUT
{attribute 'pack_mode' := '1'}
TYPE ST_RemoveStationDataIn :
STRUCT
	sCellID						: STRING(30);
	sStationID					: STRING(30);
END_STRUCT
END_TYPE

// ---- ECC/Basic/TrackClient/Method Data/Station/ST_RemoveStationDataOut.TcDUT
{attribute 'pack_mode' := '1'}
TYPE ST_RemoveStationDataOut :
STRUCT
	// Fixed data for all methods
	nNumberOfOutputArguments	: UDINT;								// determined amount of output parameters
	nReserved					: ARRAY[1..4] OF BYTE;					// Reserved padding
	
	// Method specific data
	stOutputArgInfo				: ARRAY[1..2] OF ST_UAMethodArgInfo; 	// 
	eStatus						: E_MMServerStatus;						// Status from remote method (succes/fail)
	sMessage					: STRING;								// Debugging message

END_STRUCT
END_TYPE

// ---- ECC/Basic/TrackClient/Method Data/TrafficLight/ST_AddTrafficLightData.TcDUT
TYPE ST_AddTrafficLightData :
STRUCT
	sObjectID					: STRING := 'MAIN.fbMMServer';
	sMethodID					: STRING := 'MAIN.fbMMServer#M_AddTrafficLight';
	iStatus						: INT;						// Calling status (-1: error, 0: not called, 1: calling, 2: completed OK)
	iNoOfInputArgs				: BYTE := 4;
	iNoOfOutputArgs				: BYTE := 2;
	stInput						: ST_AddTrafficLightDataIn;
	stOutput					: ST_AddTrafficLightDataOut;	
END_STRUCT
END_TYPE

// ---- ECC/Basic/TrackClient/Method Data/TrafficLight/ST_AddTrafficLightDataIn.TcDUT
{attribute 'pack_mode' := '1'}
TYPE ST_AddTrafficLightDataIn :
STRUCT
	sCellID						: STRING(30);
	sID							: STRING(30);
	iPath						: UINT;
	rPosition					: REAL;

END_STRUCT
END_TYPE

// ---- ECC/Basic/TrackClient/Method Data/TrafficLight/ST_AddTrafficLightDataOut.TcDUT
{attribute 'pack_mode' := '1'}
TYPE ST_AddTrafficLightDataOut :
STRUCT
	// Fixed data for all methods
	nNumberOfOutputArguments	: UDINT; // determined amount of output parameters
	nReserved					: ARRAY[1..4] OF BYTE; // Reserved padding
	
	// Method specific data
	stOutputArgInfo				: ARRAY[1..2] OF ST_UAMethodArgInfo; // number of output parameters - M_Mul has 1 output parameter 
	eStatus						: E_MMServerStatus;
	sMessage					: STRING;

END_STRUCT
END_TYPE

// ---- ECC/Basic/TrackClient/Method Data/TrafficLight/ST_RemoveTrafficLightData.TcDUT
TYPE ST_RemoveTrafficLightData :
STRUCT
	sObjectID					: STRING := 'MAIN.fbMMServer';
	sMethodID					: STRING := 'MAIN.fbMMServer#M_RemoveTrafficLight';
	iStatus						: INT;						// Calling status (-1: error, 0: not called, 1: calling, 2: completed OK)
	iNoOfInputArgs				: BYTE := 2;
	iNoOfOutputArgs				: BYTE := 2;
	stInput						: ST_RemoveTrafficLightDataIn;
	stOutput					: ST_RemoveTrafficLightDataOut;	
END_STRUCT
END_TYPE

// ---- ECC/Basic/TrackClient/Method Data/TrafficLight/ST_RemoveTrafficLightDataIn.TcDUT
{attribute 'pack_mode' := '1'}
TYPE ST_RemoveTrafficLightDataIn :
STRUCT
	sCellID						: STRING(30);
	sID							: STRING(30);

END_STRUCT
END_TYPE

// ---- ECC/Basic/TrackClient/Method Data/TrafficLight/ST_RemoveTrafficLightDataOut.TcDUT
{attribute 'pack_mode' := '1'}
TYPE ST_RemoveTrafficLightDataOut :
STRUCT
	// Fixed data for all methods
	nNumberOfOutputArguments	: UDINT; // determined amount of output parameters
	nReserved					: ARRAY[1..4] OF BYTE; // Reserved padding
	
	// Method specific data
	stOutputArgInfo				: ARRAY[1..2] OF ST_UAMethodArgInfo; // number of output parameters - M_Mul has 1 output parameter 
	eStatus						: E_MMServerStatus;
	sMessage					: STRING;

END_STRUCT
END_TYPE

// ---- ECC/Basic/TrackClient/Method Data/TrafficLight/ST_SetTrafficLightColorData.TcDUT
TYPE ST_SetTrafficLightColorData :
STRUCT
	sObjectID					: STRING := 'MAIN.fbMMServer';
	sMethodID					: STRING := 'MAIN.fbMMServer#M_SetTrafficLightState';
	iStatus						: INT;						// Calling status (-1: error, 0: not called, 1: calling, 2: completed OK)
	iNoOfInputArgs				: BYTE := 3;
	iNoOfOutputArgs				: BYTE := 2;
	stInput						: ST_SetTrafficLightColorDataIn;
	stOutput					: ST_SetTrafficLightColorDataOut;
END_STRUCT
END_TYPE

// ---- ECC/Basic/TrackClient/Method Data/TrafficLight/ST_SetTrafficLightColorDataIn.TcDUT
{attribute 'pack_mode' := '1'}
TYPE ST_SetTrafficLightColorDataIn :
STRUCT
	sCellID						: STRING(30);
	sID							: STRING(30);
	nColor						: INT;

END_STRUCT
END_TYPE

// ---- ECC/Basic/TrackClient/Method Data/TrafficLight/ST_SetTrafficLightColorDataOut.TcDUT
{attribute 'pack_mode' := '1'}
TYPE ST_SetTrafficLightColorDataOut :
STRUCT
	// Fixed data for all methods
	nNumberOfOutputArguments	: UDINT; // determined amount of output parameters
	nReserved					: ARRAY[1..4] OF BYTE; // Reserved padding
	
	// Method specific data
	stOutputArgInfo				: ARRAY[1..2] OF ST_UAMethodArgInfo; // number of output parameters - M_Mul has 1 output parameter 
	eStatus						: E_MMServerStatus;
	sMessage					: STRING;
	nTrafficLightState			: UINT;

END_STRUCT
END_TYPE

// ---- ECC/Basic/TrackClient/Method Data/TrafficLight/ST_TrafficLightColorData.TcDUT
TYPE ST_TrafficLightColorData :
STRUCT
	sObjectID					: STRING := 'MAIN.fbMMServer';
	sMethodID					: STRING := 'MAIN.fbMMServer#M_TrafficLightState';
	iStatus						: INT;						// Calling status (-1: error, 0: not called, 1: calling, 2: completed OK)
	iNoOfInputArgs				: BYTE := 2;
	iNoOfOutputArgs				: BYTE := 3;
	stInput						: ST_TrafficLightColorDataIn;
	stOutput					: ST_TrafficLightColorDataOut;
END_STRUCT
END_TYPE

// ---- ECC/Basic/TrackClient/Method Data/TrafficLight/ST_TrafficLightColorDataIn.TcDUT
{attribute 'pack_mode' := '1'}
TYPE ST_TrafficLightColorDataIn :
STRUCT
	sCellID						: STRING(30);
	sID							: STRING(30);

END_STRUCT
END_TYPE

// ---- ECC/Basic/TrackClient/Method Data/TrafficLight/ST_TrafficLightColorDataOut.TcDUT
{attribute 'pack_mode' := '1'}
TYPE ST_TrafficLightColorDataOut :
STRUCT
	// Fixed data for all methods
	nNumberOfOutputArguments	: UDINT; // determined amount of output parameters
	nReserved					: ARRAY[1..4] OF BYTE; // Reserved padding
	
	// Method specific data
	stOutputArgInfo				: ARRAY[1..3] OF ST_UAMethodArgInfo; // number of output parameters - M_Mul has 1 output parameter 
	eStatus						: E_MMServerStatus;
	sMessage					: STRING;
	nTrafficLightColor			: INT;

END_STRUCT
END_TYPE

// ---- ECC/Basic/TrackClient/Node Data/E_OPC_NodeType.TcDUT
{attribute 'qualified_only'}
{attribute 'strict'}
TYPE E_OPC_NodeType :
(
	Vehicles := 0,
	Paths,
	Stations,
	Cells
 
);
END_TYPE

// ---- ECC/Basic/TrackClient/Node Data/ST_ReadCellData.TcDUT
{attribute 'pack_mode' := '1'}
TYPE ST_ReadCellData :
STRUCT
	stReadListReturnInfo		: ARRAY [1..1] OF ST_UAReadListReturnInfo;
	stCell						: ST_StatusCell;

END_STRUCT
END_TYPE

// ---- ECC/Basic/TrackClient/Node Data/ST_ReadNodeData.TcDUT
{attribute 'pack_mode' := '1'}
TYPE ST_ReadNodeData :
STRUCT
	stReadListReturnInfo	: ARRAY [1..1] OF ST_UAReadListReturnInfo;
	stNodeData				: ST_StatusNode;
END_STRUCT
END_TYPE

// ---- ECC/Basic/TrackClient/Node Data/ST_ReadPathData.TcDUT
{attribute 'pack_mode' := '1'}
TYPE ST_ReadPathData :
STRUCT
	stReadListReturnInfo		: ARRAY [1..1] OF ST_UAReadListReturnInfo;
	stPathData					: ST_StatusPath;

END_STRUCT
END_TYPE

// ---- ECC/Basic/TrackClient/Node Data/ST_ReadPathData_OLD.TcDUT
{attribute 'pack_mode' := '1'}
TYPE ST_ReadPathData_OLD :
STRUCT
//	stReadListReturnInfo		: ARRAY [1..1] OF ST_UAReadListReturnInfo;
//	stPathData					: ST_StatusPath;

	// Array must have the same number as the amount of elements in the status strucuture! 
	stReadListReturnInfo		: ARRAY [1..4] OF ST_UAReadListReturnInfo;
	nPathID						: UINT;
	sCellID						: STRING(30);
	bPathPresent				: BOOL;
	nState						: UINT;
END_STRUCT
END_TYPE

